// TIA Portal project "MersinKenet200_V18" (V18)

(* hardware
DEVICE "HMI_1"  KTP900 Basic PN
   slot 0: "HMI_1"  KTP900 Basic PN  6AV2 123-2JB03-0AX0  17.0.0.0
   slot 1: "HMI_RT_1"  KTP900 Basic PN  6AV2 123-2JB03-0AX0  17.0.0.0
   slot 5: "HMI_1.IE_CP_1"  PROFINET Interface  17.0.0.0
      slot 1: "PROFINET Interface_1"  PROFINET Interface
         slot 1: "Port_1"  Port
DEVICE "S7-1200 station_1"  S7-1200 Station
   slot 0: "Rack_0"  S7-1200 Rack  Rack  V1.0
   slot 1: "PLC_1"  CPU 1214C DC/DC/DC  6ES7 214-1AG40-0XB0  V4.5
   slot 2: "DI 16/DQ 16x24VDC_1"  6ES7 223-1BL32-0XB0  V2.0
DEVICE "GSD device_1"  GSD.Device.PN
   slot 0: "Rack"  Rack  V1.0
   slot 0: "SINAMICS-V90-PN"  SINAMICS V90 PN V1.0  6SL3 210-5Fxxx-xxFx  V1.00
      slot 0: "SINAMICS V90 PN V1.0"  SINAMICS V90 PN V1.0
      slot 1: "PN-IO"  PN-IO
         slot 1: "Port 1"  Port 1
         slot 2: "Port 2"  Port 2
      slot 1: "Drive_1"  Drive
         slot 0: "Module Access Point"  Module Access Point
         slot 1: "without PROFIsafe"  without PROFIsafe
   slot 2: "SIEMENS telegram 111, PZD-12/12"  SIEMENS telegram 111, PZD-12/12
DEVICE "GSD device_2"  GSD.Device.PN
   slot 0: "Rack"  Rack  V1.0
   slot 0: "CTEU-PN"  CTEU-PN  2201471
      slot 0: "CTEU-PN"  CTEU-PN
      slot 1: "PN-IO Interface"  PN-IO Interface
         slot 1: "Port 1"  Port 1
         slot 2: "Port 2"  Port 2
   slot 1: "VAEM-L1-S-8-PT_1"  VAEM-L1-S-8-PT  573384
      slot 0: "VAEM-L1-S-8-PT"  VAEM-L1-S-8-PT
*)

// ===== PLC "PLC_1"  CPU 1214C DC/DC/DC =====

VAR_GLOBAL   // PLC tag table "Default tag table"
   "System_Byte" AT %MB1 : Byte;
   "FirstScan" AT %M1.0 : Bool;
   "DiagStatusUpdate" AT %M1.1 : Bool;
   "AlwaysTRUE" AT %M1.2 : Bool;
   "AlwaysFALSE" AT %M1.3 : Bool;
   "ManVakum" AT %M4.7 : Bool;   // Vakum pedleri manuel kontrol
   "HaziraAl_P1_Ileri" AT %M2.0 : Bool;
   "HaziraAl_P1_Geri" AT %M2.1 : Bool;
   "HaziraAl_P2_Ileri" AT %M2.2 : Bool;
   "HaziraAl_P2_Geri" AT %M2.3 : Bool;
   "HaziraAl_P3_geri" AT %M3.0 : Bool;
   "HaziraAl_ServoGoPos" AT %M3.1 : Bool;
   "ClassA_Hazir" AT %M3.2 : Bool;
   "ClassF_Hazir" AT %M3.5 : Bool;
   "ClassE_Hazir" AT %M3.3 : Bool;
   "denemeStart" AT %M3.4 : Bool;   // denemeStart
   "m50.0" AT %M3.6 : Bool;   // empty
   "AcilStop_Ris" AT %M3.7 : Bool;
   "AcilStop_Fall" AT %M5.0 : Bool;
   "empty" AT %M22.0 : Bool;
   "AutoSeq_Yesil_Lamba_Durum1" AT %M5.1 : Bool;
   "Q0.2" AT %Q0.2 : Bool;   // kirmizi lamba
   "Q0.3" AT %Q0.3 : Bool;   // sari lamba
   "Q0.4" AT %Q0.4 : Bool;   // yesil lamba
   "Q0.5" AT %Q0.5 : Bool;   // vacum
   "Q0.6" AT %Q0.6 : Bool;   // Vinc aydinlatma
   "AutoSeq_Yesil_Lamba_Durum2" AT %M5.2 : Bool;
   "Bırakma_Pos" AT %MD6 : DInt;
   "Q0.0" AT %Q0.0 : Bool;
   "Q0.1" AT %Q0.1 : Bool;
   "Q4.0" AT %Q4.0 : Bool;   // P4B-geri(kenetleme)
   "Q4.1" AT %Q4.1 : Bool;   // P4B-ileri (kenetleme)
   "Q4.2" AT %Q4.2 : Bool;   // P4-geri (kenetleme)
   "Q4.3" AT %Q4.3 : Bool;   // P4-ileri (kenetleme)
   "Q4.4" AT %Q4.4 : Bool;   // P1-geri (enayar)
   "Q4.5" AT %Q4.5 : Bool;   // P1-ileri (enayar)
   "Q4.6" AT %Q4.6 : Bool;   // P2-geri (enayar)
   "Q4.7" AT %Q4.7 : Bool;   // P2-ileri (enayar)
   "Q5.0" AT %Q5.0 : Bool;   // P3-geri (kademe)
   "Q5.1" AT %Q5.1 : Bool;   // P3-ileri (kademe)
   "ManP2_EnAyar_Ileri" AT %M5.3 : Bool;
   "ManP2_EnAyar_Geri" AT %M5.4 : Bool;
   "Gerdirme_Pos" AT %MD10 : Real;
   "AutoSeq_P3_Ileri" AT %M5.5 : Bool;
   "ManServoGoPos2" AT %M5.6 : Bool;
   "btnStartForHmi" AT %M5.7 : Bool;
   "HaziraAl_P4_P4B_Geri" AT %M14.0 : Bool;
   "MemDrive_Standsill" AT %M14.1 : Bool;
   "HaziraAl_Started" AT %M14.2 : Bool;
   "I3.6" AT %I3.6 : Bool;   // uzak kontrol cift el 2/1
   "I3.7" AT %I3.7 : Bool;   // uzak kontrol cift el 2/2
   "RemoteCiftEl" AT %M14.3 : Bool;   // Uzak kumanda cift el butonları
   "ManKenetPisP4B_Ileri" AT %M14.4 : Bool;
   "ManKenetPisP4B_Geri" AT %M14.5 : Bool;
   "vakumJenRising" AT %M14.6 : Bool;
   "Falling_Vakum_Jen" AT %M14.7 : Bool;
   "Vakum_Edge" AT %M15.0 : Bool;
   "AlarmSustur" AT %M15.1 : Bool;
END_VAR

VAR_GLOBAL   // PLC tag table "PLC"
   "Clock_Byte" AT %MB0 : Byte;
   "Clock_10Hz" AT %M0.0 : Bool;
   "Clock_5Hz" AT %M0.1 : Bool;
   "Clock_2.5Hz" AT %M0.2 : Bool;
   "Clock_2Hz" AT %M0.3 : Bool;
   "Clock_1.25Hz" AT %M0.4 : Bool;
   "Clock_1Hz" AT %M0.5 : Bool;
   "Clock_0.625Hz" AT %M0.6 : Bool;
   "Clock_0.5Hz" AT %M0.7 : Bool;
END_VAR

VAR_GLOBAL   // PLC tag table "Manuel"
   "ManServoJog1" AT %M2.4 : Bool;   // Manuel servo jog 1
   "ManServoJog2" AT %M2.5 : Bool;   // Servo manuel jog 2
   "ManServoGoHome" AT %M2.6 : Bool;   // Servo manuel go home position
   "ManServoGoPos" AT %M2.7 : Bool;   // Servo manuel kenetleme pozisyonuna git
   "ManP1_EnAyar_Ileri" AT %M4.0 : Bool;   // Manuel en ayar pistonu ileri hareket
   "ManP1_EnAyar_Geri" AT %M4.1 : Bool;   // Manuel en ayar pistonu geri hareket
   "ManKenelemePisP4_Ileri" AT %M4.2 : Bool;   // Manuel kenetleme pistonu ileri hareket
   "ManKenelemePisP4_Geri" AT %M4.3 : Bool;   // Manuel kenetleme pistonu geri hareket
   "ManKademePisIleri" AT %M4.4 : Bool;   // Manuel kademe pistonu ileri hareket
   "ManKademePisGeri" AT %M4.5 : Bool;   // Manuel kademe pistonu geri hareket
   "ManVincLambasi" AT %M4.6 : Bool;   // Vinc lambası
END_VAR

VAR_GLOBAL   // PLC tag table "Peripheral"
   "I0.0" AT %I0.0 : Bool;   // Acil Stop
   "I0.1" AT %I0.1 : Bool;   // pizzato - Cift El
   "I0.2" AT %I0.2 : Bool;   // vakum tut-bırak 1
   "I0.3" AT %I0.3 : Bool;   // vakum tut-bırak 2
   "I0.4" AT %I0.4 : Bool;   // P1 ileride
   "I0.5" AT %I0.5 : Bool;   // p1 geride
   "I0.6" AT %I0.6 : Bool;   // p1a ileride
   "I0.7" AT %I0.7 : Bool;   // p1a geride
   "I1.0" AT %I1.0 : Bool;   // p2 ileride
   "I1.1" AT %I1.1 : Bool;   // p2 geride
   "I1.2" AT %I1.2 : Bool;   // p2a ileride
   "I1.3" AT %I1.3 : Bool;   // p2a geride
   "I1.4" AT %I1.4 : Bool;   // p3 ileride
   "I1.5" AT %I1.5 : Bool;   // p3 geride
   "I2.0" AT %I2.0 : Bool;   // p3a ileride
   "I2.1" AT %I2.1 : Bool;   // p3a geride
   "I2.2" AT %I2.2 : Bool;   // p4 ileride
   "I2.3" AT %I2.3 : Bool;   // p4 geride
   "I2.4" AT %I2.4 : Bool;   // p4a ileride
   "I2.5" AT %I2.5 : Bool;   // p4a geride
   "I2.6" AT %I2.6 : Bool;   // p4b ileride
   "I2.7" AT %I2.7 : Bool;   // p4b geride
   "I3.0" AT %I3.0 : Bool;   // p4c ileride
   "I3.1" AT %I3.1 : Bool;   // p4c geride
   "I3.2" AT %I3.2 : Bool;   // lamba butonu
END_VAR

TYPE "ReceiptModel"
   STRUCT
      "Name" : String[50];   // Model Adı - 50 karakter
      Class : Int;   // Model sınıfı ( A = 0, E= 1, F = 2 )
      Boy_C : Real := 500.0;   // Model boyu (C) - mm
      En_D : Real;   // Model eni (D) - mm
   END_STRUCT;
END_TYPE

// folder: Telegram111/Receive

TYPE "ZSW1"
   STRUCT
      TolError : Bool;   // ZSW1.8 1 = Following error within tolerance
      ControlReq : Bool;   // ZSW1.9 1 = Control requested
      TarPosReached : Bool;   // ZSW1.10 1 = Target position reached
      RefPointSet : Bool;   // ZSW1.11 1 = Reference point set
      TrvTskAck : Bool;   // ZSW1.12= Acknowledgement traversing block activated
      StndStill : Bool;   // ZSW1.13 1 = This bit is used for standstill detection
      AxisAcc : Bool;   // ZSW1.14 1 = Axis accelerated
      AxisDec : Bool;   // ZSW1.15 1 = Axis decelerated
      RTS : Bool;   // ZSW1.0 1 =Ready to power up
      RDY : Bool;   // ZSW1.1 1 = Ready for operation (DC link loaded, pulses blocked)
      IOp : Bool;   // ZSW1.2 1 = Drive is switched on
      Fault : Bool;   // ZSW1.3 1 = Fault present
      OFF2Inactive : Bool;   // ZSW1.4 1 = No coast down active (OFF2 inactive)
      OFF3Inactive : Bool;   // ZSW1.5 1 = No fast stop active (OFF3 inactive)
      PowInhbt : Bool;   // ZSW1.6 1 = Activation disable active
      Alarm : Bool;   // ZSW1.7 1 = Alarm present
   END_STRUCT;
END_TYPE

TYPE "POS_ZSW1"
   STRUCT
      StopCamAct : Bool := FALSE;   // (POS_ZSW1.8) - 1 = STOP cam minus active
      StopCamPlusAct : Bool := FALSE;   // (POS_ZSW1.9) - 1 = STOP cam plus active
      jogActive : Bool := FALSE;   // (POS_ZSW1.10) - 1 = Jogging active
      ReferencePointAct : Bool := FALSE;   // (POS_ZSW1.11) - 1 = Reference point approach active
      FlyRefAct : Bool := FALSE;   // (POS_ZSW1.12) - On-the-fly homing active
      TrvBlockAct : Bool := FALSE;   // (POS_ZSW1.13) - 1 = Traversing Block active
      MdiStupAct : Bool := FALSE;   // (POS_ZSW1.14) - 1 = Set-up active
      MdiPosAct : Bool := FALSE;   // (POS_ZSW1.15) - 1 = MDI active
      Reserve : Byte;
   END_STRUCT;
END_TYPE

TYPE "POS_ZSW2"
   STRUCT
      PosActLowerCam : Bool := FALSE;   // (POS_ZSW2.8) - 1 = Position actual value ≤ cam switching position 1
      PosActGreaterCam : Bool := FALSE;   // (POS_ZSW2.9) - 1 = Position actual value ≤ cam switching position 2
      DirOut1 : Bool := FALSE;   // (POS_ZSW2.10) - 1 = Direct output 1 via traversing block
      DirOut2 : Bool := FALSE;   // (POS_ZSW2.11) - 1 = Direct output 2 via traversing block
      FixStopReached : Bool := FALSE;   // (POS_ZSW2.12) - 1 = Fixed stop reached
      FixStopTorque : Bool := FALSE;   // (POS_ZSW2.13) - 1 = Fixed stop clamping torque reached
      TravelToFixStopAct : Bool := FALSE;   // (POS_ZSW2.14) - 1 = Travel to fixed stop active
      TraversingAct : Bool := FALSE;   // (POS_ZSW2.15) - 1 = Traversing command active
      TrackingModeAct : Bool := FALSE;   // (POS_ZSW2.0) 1 = Tracking mode active
      VelocityLimAct : Bool := FALSE;   // (POS_ZSW2.1) - 1 = Velocity limiting active
      SetPStat : Bool := FALSE;   // (POS_ZSW2.2) - 1 = Setpoint set
      reserv : Bool := FALSE;   // (POS_ZSW2.3) - reserved
      MovesForward : Bool := FALSE;   // (POS_ZSW2.4) - 1 = Axis moves forward
      MovesBackward : Bool := FALSE;   // (POS_ZSW2.5) - 1 = Axis moves backwards
      SftLimSwMinReached : Bool := FALSE;   // (POS_ZSW2.6) - 1 = Software limit switch minus reached
      SftLimSwPlusReached : Bool := FALSE;   // (POS_ZSW2.7) - 1 = Software limit switch plus reached
   END_STRUCT;
END_TYPE

TYPE "ZSW2"
   STRUCT
      Reserve : Byte;
      Reserve_1 : Byte;
   END_STRUCT;
END_TYPE

TYPE "MELDW"
   STRUCT
      SpeedSetPoint : Bool;   // 1 = Speed setpoint - actual value deviation within tolerance t_on
      Reserv : Bool;
      Reserv_1 : Bool;
      ControllerEn : Bool;   // 1 = Controller enable
      DriveReady : Bool;   // MELDW.12 - 1 = Drive ready
      PulseEn : Bool;   // MELDW.13 1 = Pulses enabled
      Reserv_2 : Bool;
      Reserv_3 : Bool;
      RampFuncAct : Bool;   // MELDW.0 1 = Ramp-up/ramp-down complete 0 = Ramp-function generator active
      Reserv_4 : Bool;
      Reserv_5 : Bool;
      Reserv_6 : Bool;
      Reserv_7 : Bool;
      Reserv_8 : Bool;
      NoMotOverTemp : Bool;   // MELDW.6 1 = No motor overtemperature alarm
      NoAlrmOverload : Bool;   // MELDW.7 1 = No alarm, thermal overload, power unit
   END_STRUCT;
END_TYPE

// folder: Telegram111/Send

TYPE "STW1"
   STRUCT
      Jog1 : Bool;   // (STW1.8) - Jog 1 signal source
      Jog2 : Bool;   // (STW1.9) - Jog 2 signal source
      ControlByPlc : Bool;   // (STW1.10) - 1 = Control via PLC
      RefStart : Bool;   // (STW1.11) - 1 = Start referencing
      reserved : Bool;
      ExtBlockChange : Bool;
      reserved_1 : Bool;
      reserved_2 : Bool;
      Off1 : Bool;   // (STW1.0) - ON - 0 = OFF1 active; 1 = ON
      Off2 : Bool;   // (STW1.1) - 1 = Operating condition no coast down active
      Off3 : Bool;   // (STW1.2) - 1 = Operating condition no quick stop active
      InverterEn : Bool;   // (STW1.3) - 1 = Inverter enable
      RjcTraverTask : Bool;   // (STW1.4) - 1 = Do not reject traversing task
      IndStop : Bool;   // (STW1.5) - 1 = No intermediate stop
      TrvStart : Bool;   // (STW1.6) - Activate traversing task
      AckFaults : Bool;   // (STW1.7) - Acknowledge faults
   END_STRUCT;
END_TYPE

TYPE "POS_STW1"
   STRUCT
      MdiType : Bool;   // (POS_STW1.8) - 1 = Absolute positioning is selected 0 = Relative positioning is selected
      MdiPos : Bool;   // (POS_STW1.9) Direction selection for setting up or absolute positioning
      MdiNeg : Bool;   // (POS_STW1.10) Direction selection for setting up or absolute positioning
      reserv : Bool;
      MdiTrType : Bool;   // (POS_STW1.12) 0 = Applying values by rising edge on MdiEdge 1 = Signal: constant setpoint transfer
      reserv_1 : Bool;
      MdiSetup : Bool;   // (POS_STW1.14) => 0 = Position 1 = Setup
      MdiStart : Bool;   // (POS_STW1.15) => Operating mode MDI / direct setpoint specification
      Reserved : Byte;   // Traversing bock selection vb.
   END_STRUCT;
END_TYPE

TYPE "POS_STW2"
   STRUCT
      RefType : Bool;   // (POS_STW2.8) Homing type selection 0 = Reference point approach 1 = On-the-fly homing
      RefStartDir : Bool;   // (POS_STW2.9) - 1 = Start the search for reference in the negative direction0 = Start the search for reference in the positive direction
      RefInpS : Bool;
      RefEdge : Bool;   // (POS_STW2.11) passive homing: Setting the edge evaluation 0 = rising edge 1 = falling edge
      Reserv_3 : Bool;
      Reserv_4 : Bool;
      SftLimAct : Bool;   // (POS_STW2.14) - 1= Software limit switch activation
      StopCamAct : Bool;   // (POS_STW2.15) -1 = STOP cam active
      TrakingModeActive : Bool;   // (POS_STW2.0) -1 = Tracking mode active
      SetRefPoint : Bool;   // (POS_STW2.1) -1 = Set reference point
      ActRefCam : Bool;   // (POS_STW2.2) -1 = Reference cam active
      Reserv_5 : Bool;
      Reserv_6 : Bool;
      JogIncActv : Bool;   // (POS_STW2.5) => 0 = Continuous procedure 1 = Procedure by parameterized path
      Reserv_7 : Bool;
      Reserv_8 : Bool;
   END_STRUCT;
END_TYPE

TYPE "STW2"
   STRUCT
      Reserv : Byte;
      Reserv_1 : Byte;
   END_STRUCT;
END_TYPE

// folder: Alarm

DATA_BLOCK "Alarm_DB"   // DB9
{ S7_Optimized_Access := 'TRUE' }
VERSION : 0.1
// stored: InstanceOfName Alarm
"Alarm"
BEGIN
END_DATA_BLOCK

// folder: General

DATA_BLOCK "Out_DB"   // DB2
{ S7_Optimized_Access := 'TRUE' }
VERSION : 0.1
// stored: InstanceOfName InOut
"InOut"
BEGIN
END_DATA_BLOCK

DATA_BLOCK "HMI_Data"   // DB5
{ S7_Optimized_Access := 'TRUE' }
VERSION : 0.1
   VAR
      btnStart : Bool;
      btnStop : Bool;
      btnManuel : Bool;
      btnAuto : Bool;
      btnHaziraAl : Bool;
      EnAyarPistonu : Struct   // P1 - P2
         P1 : Struct
            btnIleri : Bool;
            btnGeri : Bool;
         END_STRUCT;
         P2 : Struct
            btnIleri : Bool;
            btnGeri : Bool;
         END_STRUCT;
      END_STRUCT;
      KenetlemePistonu : Struct   // P4-P4B
         P4 : Struct   // SAG KOLON KENETLEME
            btnIleri : Bool;
            btnGeri : Bool;
         END_STRUCT;
         P4B : Struct   // SOL KOLON KENETLEME
            btnIleri : Bool;
            btnGeri : Bool;
         END_STRUCT;
      END_STRUCT;
      "Kademe Pistonu" : Struct   // P3
         btnIleri : Bool;
         btnGeri : Bool;
      END_STRUCT;
      btnVincLambasi : Bool;
      ServoButton : Struct
         btnJogIleri : Bool;
         btnJogGeri : Bool;
         btnRefNokBelirle : Bool;
         btnHome : Bool;
         btnGoPos : Bool;
         btnHataReset : Bool;
         btnStop : Bool;   // Servo manuel işlemini durdur
         btnKenetle : Bool;   // kenetleme pozisyonuna git
      END_STRUCT;
   END_VAR
   VAR RETAIN
      ServoData : Struct
         txtActPozisyon : Real;
         txtJogOverride : Int := 100;
         txtVelocity : Real := 50.0;
         txtGerdirmeMes : Real := 10.0;   // parca gerdirme mesafesi
      END_STRUCT;
   END_VAR
   VAR
      MainInfo : String[50];
      ServoInfo : String[40];
   END_VAR
   VAR RETAIN
      KenetlemeSuresi : Time := T#1s;
   END_VAR
   VAR
      Buttons : Struct
         btnVakumJeneratoru : Bool;
         btnAlarmSustur : Bool;
      END_STRUCT;
      Status : Struct
         EnAyarPis : Struct   // P1-P1A-P2-P2A pistonları
            P1 : Struct
               Ileride : Bool;   // P1-P1A ileride
               Geride : Bool;   // P1-P1A geride
            END_STRUCT;
            P2 : Struct
               Ileride : Bool;   // P2-P2A ileride
               Geride : Bool;   // P2-P2A geride
            END_STRUCT;
         END_STRUCT;
         KademePis_P3 : Struct   // P3 pistonu
            Ileride : Bool;   // P3 pistonu ileride
            Geride : Bool;   // P3 pistonu geride
         END_STRUCT;
         KenetlemePis_P4 : Struct   // P4-P4B pistonları
            Ileride : Bool;   // P4-P4B pistonları ileride
            Geride : Bool;   // P4-P4B pistonları geride
         END_STRUCT;
      END_STRUCT;
      Alarms : Word;
      AcilSayfasi : Bool;
   END_VAR
BEGIN
END_DATA_BLOCK

DATA_BLOCK "Peripheral_Data"   // DB6
{ S7_Optimized_Access := 'TRUE' }
VERSION : 0.1
   VAR
      IN : Struct
         Acil_Stop : Bool;
         CiftEl : Struct
            IN1 : Bool;   // pizzato cift el
            IN2 : Bool;   // remote cift el 1
            IN3 : Bool;   // remote cift el 2
         END_STRUCT;
         EnAyar : Struct   // P1,P1A,P2,P2A
            P1 : Struct
               Ileride : Bool;
               Geride : Bool;
            END_STRUCT;
            P1A : Struct
               Ileride : Bool;
               Geride : Bool;
            END_STRUCT;
            P2 : Struct
               Ileride : Bool;
               Geride : Bool;
            END_STRUCT;
            P2A : Struct
               Ileride : Bool;
               Geride : Bool;
            END_STRUCT;
         END_STRUCT;
         KademeAyar : Struct   // P3,P3A
            P3 : Struct
               Ileride : Bool;
               Geride : Bool;
            END_STRUCT;
         END_STRUCT;
         Kenetleme : Struct   // P4,P4A,P4B,P4C
            P4 : Struct
               Ilderide : Bool;
               Geride : Bool;
            END_STRUCT;
            P4B : Struct
               Ilderide : Bool;
               Geride : Bool;
            END_STRUCT;
         END_STRUCT;
         VincUstuLamba : Bool;
         VakumJen : Bool;
         ServoHomeSen : Bool;   // Servo home sensoru
      END_STRUCT;
      OUT : Struct
         EnAyar : Struct   // P1,P1A,P2,P2A
            P1 : Struct
               Ileri : Bool;
               Geri : Bool;
            END_STRUCT;
            P2 : Struct
               Ileri : Bool;
               Geri : Bool;
            END_STRUCT;
         END_STRUCT;
         KademeAyar : Struct   // P3,P3A
            P3 : Struct
               Ileri : Bool;
               Geri : Bool;
            END_STRUCT;
         END_STRUCT;
         Kenetleme : Struct   // P4,P4A,P4B,P4C
            P4_P4A : Struct
               Ilderi : Bool;
               Geri : Bool;
            END_STRUCT;
            P4B_P4C : Struct
               Ilderi : Bool;
               Geri : Bool;
            END_STRUCT;
         END_STRUCT;
         LAMBA : Struct
            Yesil : Bool;
            Kirmizi : Bool;
            Sari : Bool;
            Buzzer : Bool;
         END_STRUCT;
         VincLambasi : Bool;
         Vacum : Bool;   // Vakum jeneratoru
      END_STRUCT;
   END_VAR
BEGIN
END_DATA_BLOCK

DATA_BLOCK "System_Data"   // DB7
{ S7_Optimized_Access := 'TRUE' }
VERSION : 0.1
   VAR
      AutoSeq_State : Int;
      AutoSeq_Busy : Bool;
      AutoSeq_Done : Bool;
      AutoSeq_Message : String[50];
      Ready : Bool;
      CmdDrive : Struct
         GoPos : Bool;
         GoHome : Bool;
         SetReference : Bool;
         Jog1 : Bool;
         Jog2 : Bool;
         Position : Real;
         Velocity : Real;
         Override : Int;
         AckError : Bool;
         Message : String[40];
         Pos_Done : Bool;
         Busy : Bool;
         Error : Bool;
         AxisError : Bool;
         ErrorId : Byte;
         ReferencedAxis : Bool;
         ActPosition : Real;
         HomePosition : Real;   // Servo durması gereken home pozisyonu
         Alarm : Word;
         IsHomePosTol : Bool;   // Axis home konumu tolerans icinde
         IsPosTol : Bool;   // Axis pozisyon konumu tolerans icinde
      END_STRUCT;
      SystemMode : Struct
         Auto : Bool;
         Man : Bool;
      END_STRUCT;
      AutoSeq : Struct
         GoPos : Bool;   // Parça kenetleme
         GoPos2 : Bool;   // Parça birakma
         GoHome : Bool;
         P3_Ileri : Bool;
         P3_Geri : Bool;   // kademe pistonu
         "P4-P4A_Ileri" : Bool;   // kenetleme pistonu
         "P4-P4A_geri" : Bool;
         "P4B-P4C_Ileri" : Bool;
         StartedInfo : Bool;   // otomatik mod basladi
      END_STRUCT;
   END_VAR
BEGIN
END_DATA_BLOCK

DATA_BLOCK "SINA_POS_DB"   // DB11
{ S7_Optimized_Access := 'TRUE' }
AUTHOR : DRVDPS7
FAMILY : DRIVES
NAME : SINA_POS
VERSION : 5.7
// stored: InstanceOfName SINA_POS
"SINA_POS"
BEGIN
END_DATA_BLOCK

// folder: Manuel

DATA_BLOCK "Manuel_DB"   // DB4
{ S7_Optimized_Access := 'TRUE' }
VERSION : 0.1
// stored: InstanceOfName Manuel
"Manuel"
BEGIN
END_DATA_BLOCK

// folder: Otomatik

DATA_BLOCK "Otomatik_Seq_LAD_DB"   // DB8
{ S7_Optimized_Access := 'TRUE' }
VERSION : 0.1
// stored: InstanceOfName Otomatik_Seq_LAD
"Otomatik_Seq_LAD"
BEGIN
END_DATA_BLOCK

// folder: Receipt

DATA_BLOCK "Receipt"   // DB1
{ S7_Optimized_Access := 'TRUE' }
VERSION : 0.1
   VAR RETAIN
      ModelId : Int;   // Combobox index numarasi
      OldModelId : Int;
      ModelList : Array[0..25] of "ReceiptModel";   // Model listesi
      CurrentModel : "ReceiptModel";   // Secili model
   END_VAR
   VAR
      btnSave : Bool;   // Recete kaydet butonu - HMI
      bShowMessage : Bool;   // Kaydedildi mesaji icin
      tSavedTimer : IEC_TIMER;
   END_VAR
BEGIN
END_DATA_BLOCK

// folder: (top level)

ORGANIZATION_BLOCK "Task_1"   // OB1, LAD, ProgramCycle
TITLE = "Main Program Sweep (Cycle)"
{ S7_Optimized_Access := 'TRUE' }
VERSION : 0.1
   VAR_INPUT
      Initial_Call : Bool;   // Initial call of this OB
      Remanence : Bool;   // =True, if remanent data are available
   END_VAR
   VAR_TEMP
      bSeqStart : Bool;   // Otomatik sekans baslat
   END_VAR
BEGIN

REGION Network 1: Sistem acildiginda ilk cycle ile manuel setle (bir seferlik calisir)
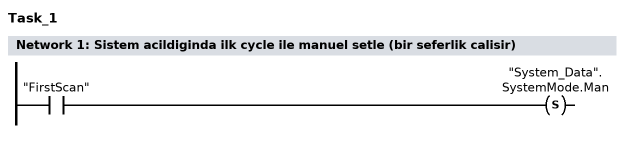
   RUNG wire#powerrail
      Contact( "FirstScan" )
      S_Coil( "System_Data".SystemMode.Man )
   END_RUNG
   // the same network as SCL:
   IF "FirstScan" THEN "System_Data".SystemMode.Man := TRUE; END_IF;
END_REGION

REGION Network 2 (SCL): Otomatik sekans baslat
   "Peripheral"();
   "Out_DB"();
   "Station"();

   #bSeqStart := "Peripheral_Data".IN.CiftEl.IN1 AND "RemoteCiftEl";
   "Otomatik_Seq_LAD_DB"(Start := #bSeqStart,
                         //Start := "btnStartForHmi",
                         Stop := "HMI_Data".btnStop,
                         EmergencyStop := "Peripheral_Data".IN.Acil_Stop,
                         Busy => "System_Data".AutoSeq_Busy,
                         Done => "System_Data".AutoSeq_Done,
                         Message => "System_Data".AutoSeq_Message);
END_REGION
END_ORGANIZATION_BLOCK

ORGANIZATION_BLOCK "Hardware interrupt"   // OB40, LAD, HWProcessInterrupt
{ S7_Optimized_Access := 'TRUE' }
VERSION : 0.1
   VAR_INPUT
      LADDR : Hw_Io;   // Hardware identifier
      USI : Word;   // User structure identifier
      IChannel : USInt;   // Interrupt channel number
      EventType : Byte;   // EventType
   END_VAR
BEGIN
END_ORGANIZATION_BLOCK

ORGANIZATION_BLOCK "Diagnostic error interrupt"   // OB82, LAD, DiagnosticErrorInterrupt
{ S7_Optimized_Access := 'TRUE' }
VERSION : 0.1
   VAR_INPUT
      IO_State : Word;   // IO state of the HW object
      LADDR : Hw_Any;   // Hardware identifier
      Channel : UInt;   // Channel number
      MultiError : Bool;   // =true if more than one error is present
   END_VAR
BEGIN
END_ORGANIZATION_BLOCK

ORGANIZATION_BLOCK "Pull or plug of modules"   // OB83, LAD, PullPlug
{ S7_Optimized_Access := 'TRUE' }
VERSION : 0.1
   VAR_INPUT
      LADDR : Hw_Io;   // Hardware identifier
      Event_Class : Byte;   // 16#38/39: module inserted, removed
      Fault_ID : Byte;   // Fault identifier
   END_VAR
BEGIN
END_ORGANIZATION_BLOCK

ORGANIZATION_BLOCK "Rack or station failure"   // OB86, LAD, RackStationFailure
{ S7_Optimized_Access := 'TRUE' }
VERSION : 0.1
   VAR_INPUT
      LADDR : Hw_Device;   // Hardware identifier
      Event_Class : Byte;   // Event class
      Fault_ID : Byte;   // Fault identifier
   END_VAR
BEGIN
END_ORGANIZATION_BLOCK

ORGANIZATION_BLOCK "Startup"   // OB100, LAD, Startup
TITLE = "Complete Restart"
{ S7_Optimized_Access := 'TRUE' }
VERSION : 0.1
   VAR_INPUT
      LostRetentive : Bool;   // True if retentive data are lost
      LostRTC : Bool;   // True if date and time are lost
   END_VAR
BEGIN

REGION Network 1
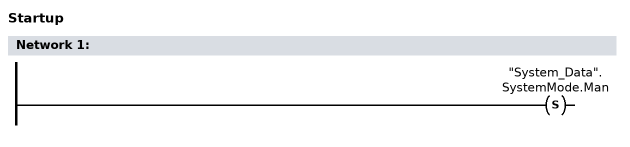
   RUNG wire#powerrail
      S_Coil( "System_Data".SystemMode.Man )
   END_RUNG
   // the same network as SCL:
   "System_Data".SystemMode.Man := TRUE;
END_REGION
END_ORGANIZATION_BLOCK

ORGANIZATION_BLOCK "Task_2"   // OB123, LAD, ProgramCycle
TITLE = "Main Program Sweep (Cycle)"
{ S7_Optimized_Access := 'TRUE' }
VERSION : 0.1
   VAR_INPUT
      Initial_Call : Bool;   // Initial call of this OB
      Remanence : Bool;   // =True, if remanent data are available
   END_VAR
BEGIN

REGION Network 2 (SCL)
   "ReceiptManager"();
   "Manuel_DB"();
   "HMI"();
   "HaziraAl"(Execute:="HMI_Data".btnHaziraAl,
              EmergencyStop:="Peripheral_Data".IN.Acil_Stop,
              IsServoPosDone:="System_Data".CmdDrive.Pos_Done,
              Manuel:="System_Data".SystemMode.Man,
              AxisReferenced:="System_Data".CmdDrive.ReferencedAxis,
              P1_Ileri=>"HaziraAl_P1_Ileri",
              P1_Geri=>"HaziraAl_P1_Geri",
              P2_Ileri=>"HaziraAl_P2_Ileri",
              P2_geri=>"HaziraAl_P2_Geri",
              P3_geri=>"HaziraAl_P3_geri",
              P4_P4B_Geri=>"HaziraAl_P4_P4B_Geri",
              ServoGoPos=>"HaziraAl_ServoGoPos",
              ClassA_Hazir=>"ClassA_Hazir",
              ClassE_Hazir=>"ClassE_Hazir",
              ClassF_Hazir=>"ClassF_Hazir");

   "Alarm_DB"();
   "UyariLambasi"();
END_REGION
END_ORGANIZATION_BLOCK

// folder: Alarm

FUNCTION_BLOCK "Alarm"   // FB7, LAD
{ S7_Optimized_Access := 'TRUE' }
VERSION : 0.1
   VAR
      timeInterval : Time;
      p1_ileri_Timer : TON_TIME;
      p1_geri_Timer : TON_TIME;
      p2_Ileri_Timer : TON_TIME;
      p2_geri_Timer : TON_TIME;
      p3_ileri_Timer : TON_TIME;
      p3_geri_Timer : TON_TIME;
      p4_ileri_Timer : TON_TIME;
      p4_geri_Timer : TON_TIME;
      p4b_ileri_Timer : TON_TIME;
      p4b_geri_Timer : TON_TIME;
      wAlarmsServoOrCylinder : Word;
      wAlarmsPeripheral : Word;
   END_VAR
BEGIN

REGION Network 1: timer interval
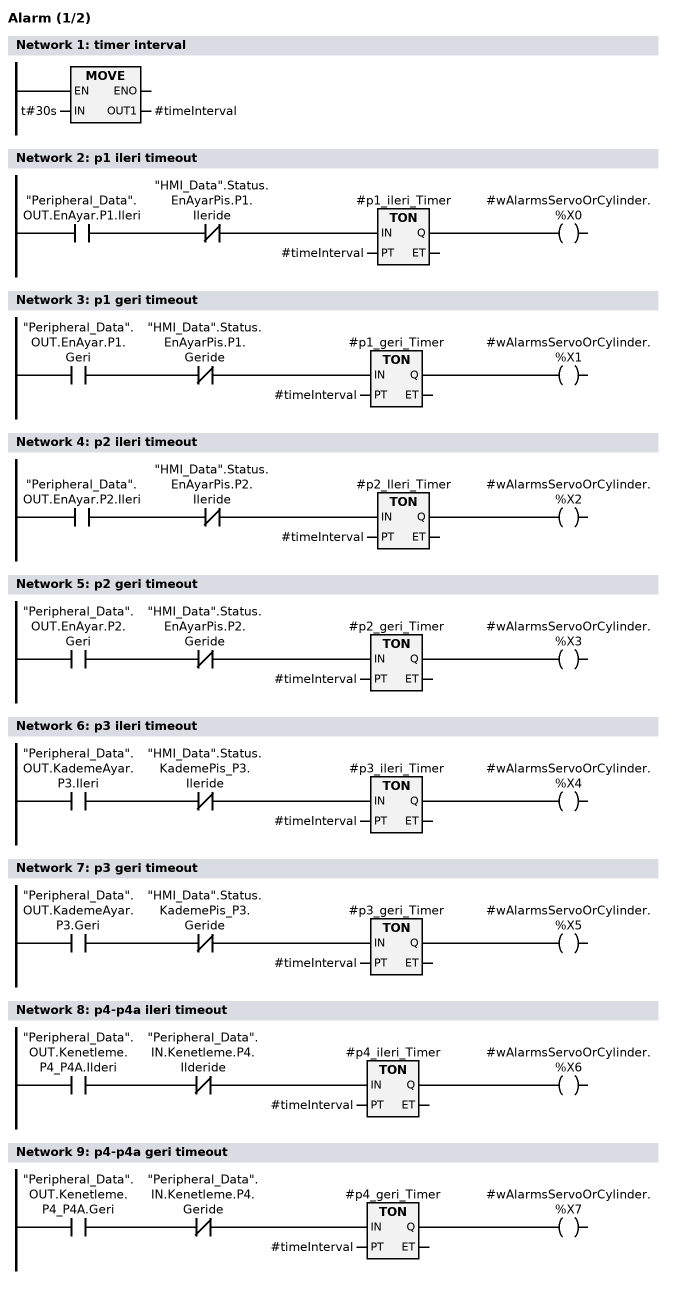
   RUNG wire#powerrail
      Move(in := t#30s, out1 => #timeInterval)
   END_RUNG
   // the same network as SCL:
   #timeInterval := t#30s;
END_REGION

REGION Network 2: p1 ileri timeout
   #p1_ileri_Timer(IN := "Peripheral_Data".OUT.EnAyar.P1.Ileri AND NOT "HMI_Data".Status.EnAyarPis.P1.Ileride,   // TON
                   PT := #timeInterval);
   #wAlarmsServoOrCylinder.%X0 := #p1_ileri_Timer.Q;
END_REGION

REGION Network 3: p1 geri timeout
   #p1_geri_Timer(IN := "Peripheral_Data".OUT.EnAyar.P1.Geri AND NOT "HMI_Data".Status.EnAyarPis.P1.Geride,   // TON
                  PT := #timeInterval);
   #wAlarmsServoOrCylinder.%X1 := #p1_geri_Timer.Q;
END_REGION

REGION Network 4: p2 ileri timeout
   #p2_Ileri_Timer(IN := "Peripheral_Data".OUT.EnAyar.P2.Ileri AND NOT "HMI_Data".Status.EnAyarPis.P2.Ileride,   // TON
                   PT := #timeInterval);
   #wAlarmsServoOrCylinder.%X2 := #p2_Ileri_Timer.Q;
END_REGION

REGION Network 5: p2 geri timeout
   #p2_geri_Timer(IN := "Peripheral_Data".OUT.EnAyar.P2.Geri AND NOT "HMI_Data".Status.EnAyarPis.P2.Geride,   // TON
                  PT := #timeInterval);
   #wAlarmsServoOrCylinder.%X3 := #p2_geri_Timer.Q;
END_REGION

REGION Network 6: p3 ileri timeout
   #p3_ileri_Timer(IN := "Peripheral_Data".OUT.KademeAyar.P3.Ileri AND NOT "HMI_Data".Status.KademePis_P3.Ileride,   // TON
                   PT := #timeInterval);
   #wAlarmsServoOrCylinder.%X4 := #p3_ileri_Timer.Q;
END_REGION

REGION Network 7: p3 geri timeout
   #p3_geri_Timer(IN := "Peripheral_Data".OUT.KademeAyar.P3.Geri AND NOT "HMI_Data".Status.KademePis_P3.Geride,   // TON
                  PT := #timeInterval);
   #wAlarmsServoOrCylinder.%X5 := #p3_geri_Timer.Q;
END_REGION

REGION Network 8: p4-p4a ileri timeout
   #p4_ileri_Timer(IN := "Peripheral_Data".OUT.Kenetleme.P4_P4A.Ilderi AND NOT "Peripheral_Data".IN.Kenetleme.P4.Ilderide,   // TON
                   PT := #timeInterval);
   #wAlarmsServoOrCylinder.%X6 := #p4_ileri_Timer.Q;
END_REGION

REGION Network 9: p4-p4a geri timeout
   #p4_geri_Timer(IN := "Peripheral_Data".OUT.Kenetleme.P4_P4A.Geri AND NOT "Peripheral_Data".IN.Kenetleme.P4.Geride,   // TON
                  PT := #timeInterval);
   #wAlarmsServoOrCylinder.%X7 := #p4_geri_Timer.Q;
END_REGION

REGION Network 10: p4b-p4c ileri timeout
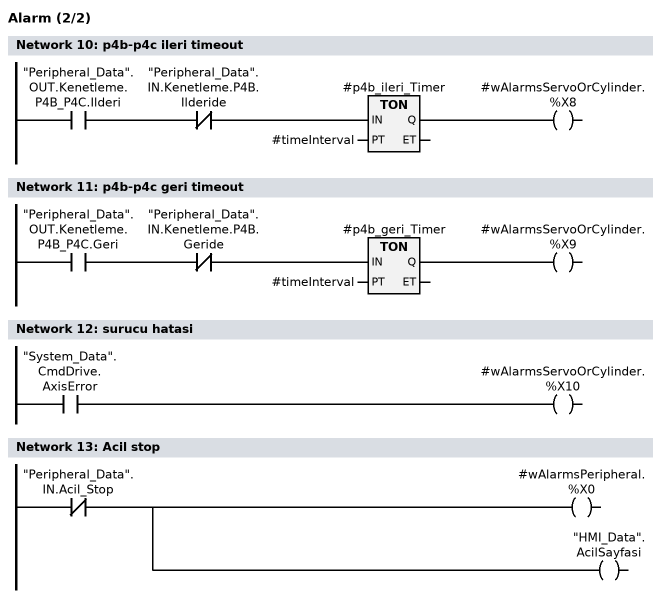
   #p4b_ileri_Timer(IN := "Peripheral_Data".OUT.Kenetleme.P4B_P4C.Ilderi AND NOT "Peripheral_Data".IN.Kenetleme.P4B.Ilderide,   // TON
                    PT := #timeInterval);
   #wAlarmsServoOrCylinder.%X8 := #p4b_ileri_Timer.Q;
END_REGION

REGION Network 11: p4b-p4c geri timeout
   #p4b_geri_Timer(IN := "Peripheral_Data".OUT.Kenetleme.P4B_P4C.Geri AND NOT "Peripheral_Data".IN.Kenetleme.P4B.Geride,   // TON
                   PT := #timeInterval);
   #wAlarmsServoOrCylinder.%X9 := #p4b_geri_Timer.Q;
END_REGION

REGION Network 12: surucu hatasi
   RUNG wire#powerrail
      Contact( "System_Data".CmdDrive.AxisError )
      Coil( #wAlarmsServoOrCylinder.%X10 )
   END_RUNG
   // the same network as SCL:
   #wAlarmsServoOrCylinder.%X10 := "System_Data".CmdDrive.AxisError;
END_REGION

REGION Network 13: Acil stop
   RUNG wire#powerrail
      I_Contact( "Peripheral_Data".IN.Acil_Stop )
      wire#w1
      Coil( #wAlarmsPeripheral.%X0 )
   END_RUNG
   RUNG wire#w1
      Coil( "HMI_Data".AcilSayfasi )
   END_RUNG
   // the same network as SCL:
   #wAlarmsPeripheral.%X0 := NOT "Peripheral_Data".IN.Acil_Stop;
   "HMI_Data".AcilSayfasi := NOT "Peripheral_Data".IN.Acil_Stop;
END_REGION
END_FUNCTION_BLOCK

// folder: BaseClass

FUNCTION_BLOCK "CiftEl"   // FB11, LAD
{ S7_Optimized_Access := 'TRUE' }
VERSION : 0.1
   VAR_INPUT
      In_1 : Bool;   // Cift el
      In_2 : Bool;   // Cift el
   END_VAR
   VAR_OUTPUT
      Out : Bool;   // out
   END_VAR
   VAR
      IEC_Timer_0_Instance : TP_TIME;
      IEC_Timer_0_Instance_1 : TP_TIME;
      IEC_Timer_0_Instance_2 : TOF_TIME;
      stOut : Bool;
   END_VAR
   VAR_TEMP
      bCiftEl_1 : Bool;
      bCiftEl_2 : Bool;
   END_VAR
BEGIN

REGION Network 1
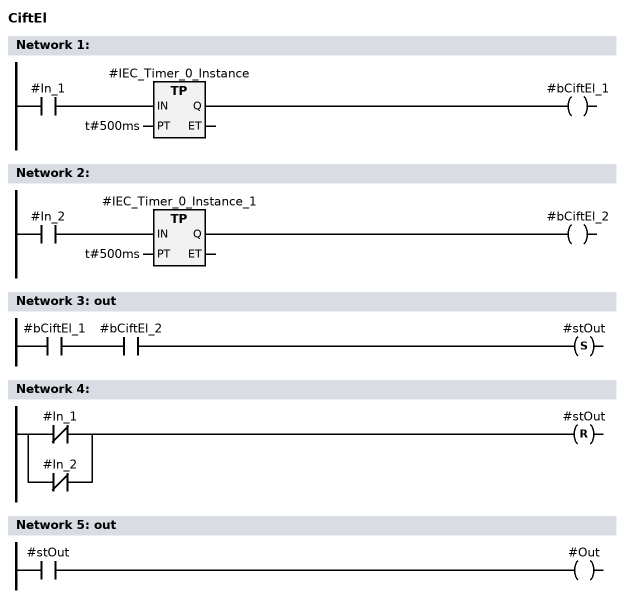
   #IEC_Timer_0_Instance(IN := #In_1, PT := t#500ms);   // TP
   #bCiftEl_1 := #IEC_Timer_0_Instance.Q;
END_REGION

REGION Network 2
   #IEC_Timer_0_Instance_1(IN := #In_2, PT := t#500ms);   // TP
   #bCiftEl_2 := #IEC_Timer_0_Instance_1.Q;
END_REGION

REGION Network 3: out
   RUNG wire#powerrail
      Contact( #bCiftEl_1 )
      Contact( #bCiftEl_2 )
      S_Coil( #stOut )
   END_RUNG
   // the same network as SCL:
   IF #bCiftEl_1 AND #bCiftEl_2 THEN #stOut := TRUE; END_IF;
END_REGION

REGION Network 4
   RUNG wire#powerrail
      I_Contact( #In_1 )
      wire#w1
      R_Coil( #stOut )
   END_RUNG
   RUNG wire#powerrail
      I_Contact( #In_2 )
   END_RUNG wire#w1
   // the same network as SCL:
   IF NOT #In_1 OR NOT #In_2 THEN #stOut := FALSE; END_IF;
END_REGION

REGION Network 5: out
   RUNG wire#powerrail
      Contact( #stOut )
      Coil( #Out )
   END_RUNG
   // the same network as SCL:
   #Out := #stOut;
END_REGION
END_FUNCTION_BLOCK

// folder: BaseClass/Drive

FUNCTION_BLOCK "BaseDrive_LAD"   // FB10, LAD
{ S7_Optimized_Access := 'TRUE' }
VERSION : 0.1
   VAR_INPUT
      Enable : Bool;   // BaseDrive enable
      Emergency : Bool;   // acil stop
      GoPos : Bool;   // kenetleme pozisyonuna git
      SetReference : Bool;   // referans ayarla
      Jog1 : Bool;   // servo jog 1 - negatif yon
      Jog2 : Bool;   // servo jog 1 - positive yon
      Position : Real;   // model kenetleme konumu
      Velocity : Real := 50.0;   // % (0 - 100) arası
      Override : Int := 100;   // % (0 - 100) arası
      AckError : Bool;   // servo hata reset
      HWDSTW : Hw_Io;
      HWDZSW : Hw_Io;
   END_VAR
   VAR_OUTPUT
      Pos_Done : Bool;
      Busy : Bool;
      Error : Bool;
      AxisError : Bool;   // Axis hatasi
      ErrorId : Byte;
      ReferencedAxis : Bool;   // reference point set
      Message : String[40];
      ActPosition : Real;
      Alarm : Word;   // Drive hataları
      IsPosTol : Bool;   // Axis pozisyon konumu tolerans icinde
      Standstill : Bool;   // servo durdu
   END_VAR
   VAR
      SINA_POS_Instance_1 : "SINA_POS";
      stState : Int;
      stMdiMode : Int;
      stEnableAxis : Bool;
      stTargetPos : DInt;
      stVelocity : DInt;
      stExecute : Bool;
      stAxisPosDone : Bool;
      stAxisError : Bool;
      IsDoneDelay : TON_TIME;
      DelayMessage : TON_TIME;
      IsDoneDelay_IN : Bool;
      IsDoneDelay_Q : Bool;
      DelayMessage_IN : Bool;
      DelayMessage_Q : Bool;
      stOverride : Int;
      stActualPosition : DInt;
      stHomingMode : Int;
      stHomingError : Bool;
      stHomingErrorId : Word;
      bHomingRefOk : Bool;
      stActualVelocity : DInt;
      DelayOnOff1_1 : TON_TIME;
      DelayOnOff1_2 : TON_TIME;
      DelayOnOff1_1_IN : Bool;
      DelayOnOff1_1_Q : Bool;
      DelayOnOff1_2_IN : Bool;
      DelayOnOff1_2_Q : Bool;
      stRefOk : Bool;   // Referans tanımlandı
      stPositionMax : DInt;
      stPositionMin : DInt;
      stConfigEpos : DWord;
      stEposZsw2 : Word;
      stPositive : Bool;   // referans bulma yonu
      stAxisEnabled : Bool;   // OFF1 geldikten sonra setlenir
      Toff1_Instance : TOF_TIME;
      Toff1_IN : Bool;
      Toff1_Q : Bool;
   END_VAR
   VAR_TEMP
      dnPosition : DInt;
      bJog1 : Bool;
      bJog2 : Bool;
      bGoPos : Bool;
      bSetReference : Bool;
      bBusy : Bool;
      bError : Bool;
      bPosDone : Bool;
      rVelocity : Real;
      rOverride : Int;
      nOverride : Int;
      bHomingOff1 : Bool;
      bHomingExecute : Bool;
      bHomingHWLimitActive : Bool;
      bAckError : Bool;
      wAlarm : Word;
      bStandstill : Bool;
   END_VAR
   VAR CONSTANT
      eIDLE : Int := 0;
      eGOPOS_PRE : Int := 1;
      eGOPOS_RUN : Int := 2;
      eREFERENCE_PRE : Int := 3;
      eREFERENCE_RUN : Int := 4;
      eJOG_RUN : Int := 5;
      eJOG_POSITIVE : Int := 6;
      eSUCCESS : Int := 7;
      eERROR : Int := 8;
      eInterrupt : Int := 11;
      eMessage : Int := 12;
      eAxisError : Int := 13;
      eRESET : Int := 14;
   END_VAR
   VAR_TEMP   // added for the SCL form of the ladder/FBD networks
      _w1 : Bool;
      _w2 : Bool;
   END_VAR
BEGIN

REGION Network 2 (SCL): Tanımlamalar
   REGION "TIMER" 
       #IsDoneDelay(IN := #IsDoneDelay_IN,
                    PT := t#400ms,
                    Q => #IsDoneDelay_Q);

       #DelayOnOff1_1(IN := #DelayOnOff1_1_IN,
                      PT := T#300MS,
                      Q => #DelayOnOff1_1_Q);

       #DelayOnOff1_2(IN := #DelayOnOff1_2_IN,
                      PT := T#300MS,
                      Q => #DelayOnOff1_2_Q);

       #Toff1_Instance(IN := #Toff1_IN,
                       PT := t#500ms,
                       Q => #Toff1_Q);
   END_REGION

   REGION "LOCAL DEGISKENLER" 
   (*
       N/M = 1/1 ise 
       PER REVOLUTION = 10000 ise
       BİR TURDA 10mm gider
       Ekrandan gelen pozisyon değerini bin ile çarpılır.
   *)
       #bGoPos := #GoPos;
       #dnPosition := REAL_TO_DINT( #Position * 1000.0 );  // 10000 LU -> 10 mm yapıyor
       #bSetReference := #SetReference;
       #bAckError := #stAxisError AND #AckError;

       #DelayOnOff1_1_IN := NOT #stAxisError AND #Enable;

       #stEnableAxis := #DelayOnOff1_1_Q AND #Enable;

       // #Toff1_IN := #DelayOnOff1_1_Q AND #Enable;
       // #stEnableAxis := #Toff1_Q;

   END_REGION

   REGION "Posizyon Tolerans"

       #stPositionMax := #dnPosition + 4000;
       #stPositionMin := #dnPosition - 4000;

       #IsPosTol := #SINA_POS_Instance_1.ActPosition > #stPositionMin
       AND #SINA_POS_Instance_1.ActPosition < #stPositionMax;

   END_REGION

   REGION "YUZDELIK HIZ HESABI"
       #rVelocity := (#Velocity * 16384.0) / 100.0;
       #stVelocity := REAL_TO_DINT(#rVelocity);  // Hiz bilgisini yukle

   END_REGION

   REGION "JOG HIZ AYARI" 

       #stOverride := #Override;

   END_REGION
END_REGION

REGION Network 3: Baslangic adimi
   // Bos adim
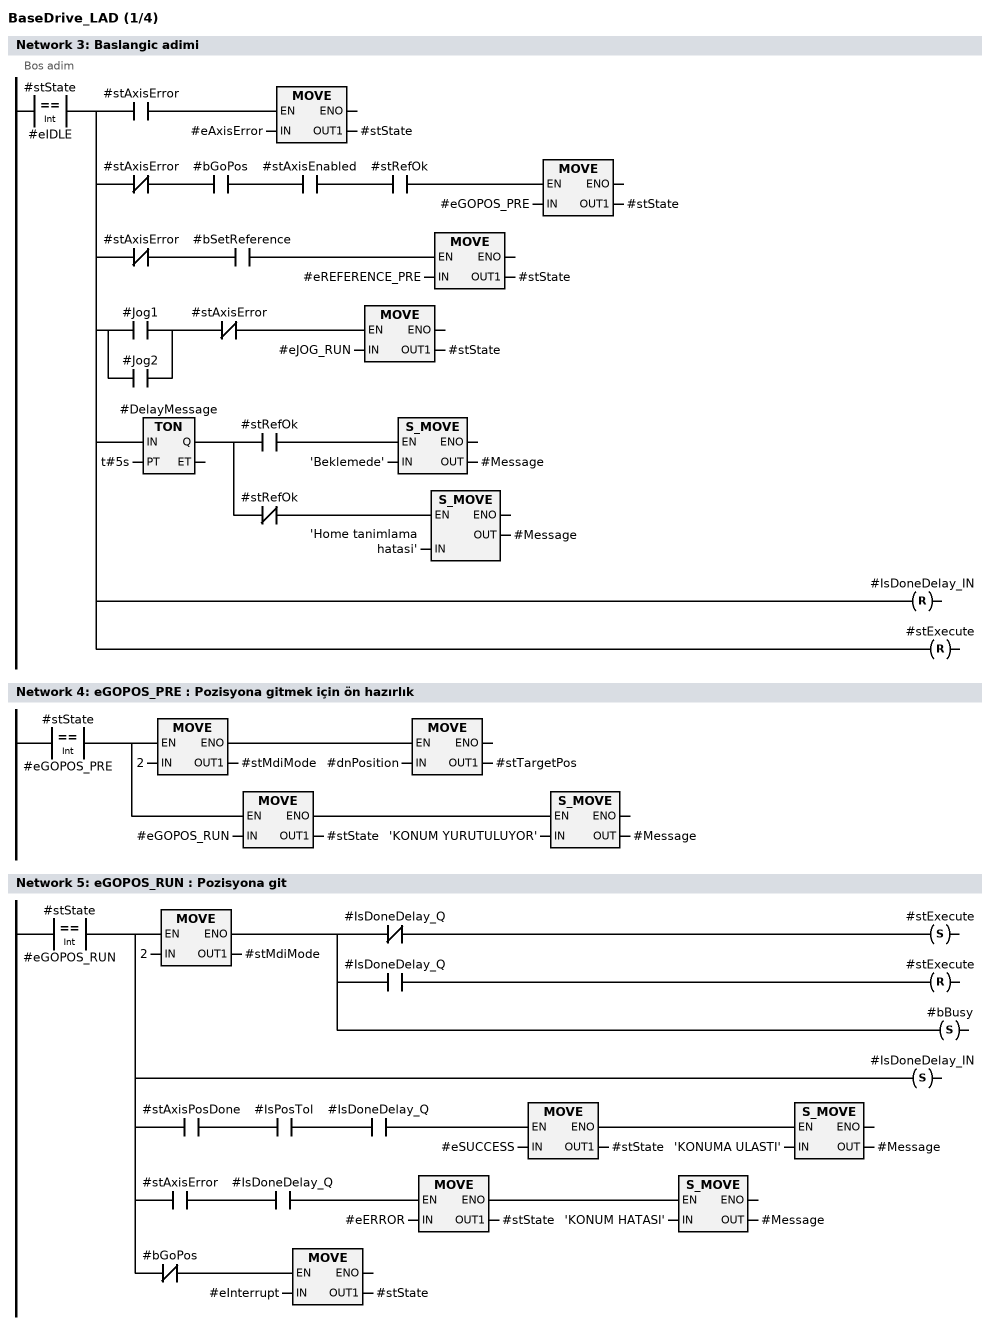
   #_w1 := #stState = #eIDLE;
   IF #_w1 AND #stAxisError THEN #stState := #eAxisError; END_IF;
   IF #_w1 AND NOT #stAxisError AND #bGoPos AND #stAxisEnabled AND #stRefOk THEN
       #stState := #eGOPOS_PRE;
   END_IF;
   IF #_w1 AND NOT #stAxisError AND #bSetReference THEN #stState := #eREFERENCE_PRE; END_IF;
   IF #_w1 AND (#Jog1 OR #Jog2) AND NOT #stAxisError THEN #stState := #eJOG_RUN; END_IF;
   #DelayMessage(IN := #_w1, PT := t#5s);   // TON
   IF #DelayMessage.Q AND #stRefOk THEN #Message := 'Beklemede'; END_IF;
   IF #DelayMessage.Q AND NOT #stRefOk THEN #Message := 'Home tanimlama hatasi'; END_IF;
   IF #_w1 THEN
       #IsDoneDelay_IN := FALSE;
       #stExecute := FALSE;
   END_IF;
END_REGION

REGION Network 4: eGOPOS_PRE : Pozisyona gitmek için ön hazırlık
   RUNG wire#powerrail
      { S7_Templates := "SrcType := Int" } EQ_Contact(in1 := #stState, in2 := #eGOPOS_PRE)
      wire#w1
      Move(in := 2, out1 => #stMdiMode)
      Move(in := #dnPosition, out1 => #stTargetPos)
   END_RUNG
   RUNG wire#w1
      Move(in := #eGOPOS_RUN, out1 => #stState)
      S_Move(in := 'KONUM YURUTULUYOR', out => #Message)
   END_RUNG
   // the same network as SCL:
   IF #stState = #eGOPOS_PRE THEN
       #stMdiMode := 2;
       #stTargetPos := #dnPosition;
   END_IF;
   #_w1 := #stState = #eGOPOS_PRE;
   IF #_w1 THEN
       #stState := #eGOPOS_RUN;
       #Message := 'KONUM YURUTULUYOR';
   END_IF;
END_REGION

REGION Network 5: eGOPOS_RUN : Pozisyona git
   RUNG wire#powerrail
      { S7_Templates := "SrcType := Int" } EQ_Contact(in1 := #stState, in2 := #eGOPOS_RUN)
      wire#w1
      Move(in := 2, out1 => #stMdiMode)
      wire#w2
      I_Contact( #IsDoneDelay_Q )
      S_Coil( #stExecute )
   END_RUNG
   RUNG wire#w2
      Contact( #IsDoneDelay_Q )
      R_Coil( #stExecute )
   END_RUNG
   RUNG wire#w2
      S_Coil( #bBusy )
   END_RUNG
   RUNG wire#w1
      S_Coil( #IsDoneDelay_IN )
   END_RUNG
   RUNG wire#w1
      Contact( #stAxisPosDone )
      Contact( #IsPosTol )
      Contact( #IsDoneDelay_Q )
      Move(in := #eSUCCESS, out1 => #stState)
      S_Move(in := 'KONUMA ULASTI', out => #Message)
   END_RUNG
   RUNG wire#w1
      Contact( #stAxisError )
      Contact( #IsDoneDelay_Q )
      Move(in := #eERROR, out1 => #stState)
      S_Move(in := 'KONUM HATASI', out => #Message)
   END_RUNG
   RUNG wire#w1
      I_Contact( #bGoPos )
      Move(in := #eInterrupt, out1 => #stState)
   END_RUNG
   // the same network as SCL:
   #_w1 := #stState = #eGOPOS_RUN;
   IF #_w1 THEN #stMdiMode := 2; END_IF;
   IF #_w1 AND NOT #IsDoneDelay_Q THEN #stExecute := TRUE; END_IF;
   IF #_w1 AND #IsDoneDelay_Q THEN #stExecute := FALSE; END_IF;
   IF #_w1 THEN
       #bBusy := TRUE;
       #IsDoneDelay_IN := TRUE;
   END_IF;
   IF #_w1 AND #stAxisPosDone AND #IsPosTol AND #IsDoneDelay_Q THEN
       #stState := #eSUCCESS;
       #Message := 'KONUMA ULASTI';
   END_IF;
   IF #_w1 AND #stAxisError AND #IsDoneDelay_Q THEN
       #stState := #eERROR;
       #Message := 'KONUM HATASI';
   END_IF;
   IF #_w1 AND NOT #bGoPos THEN #stState := #eInterrupt; END_IF;
END_REGION

REGION Network 6: Referans belirle
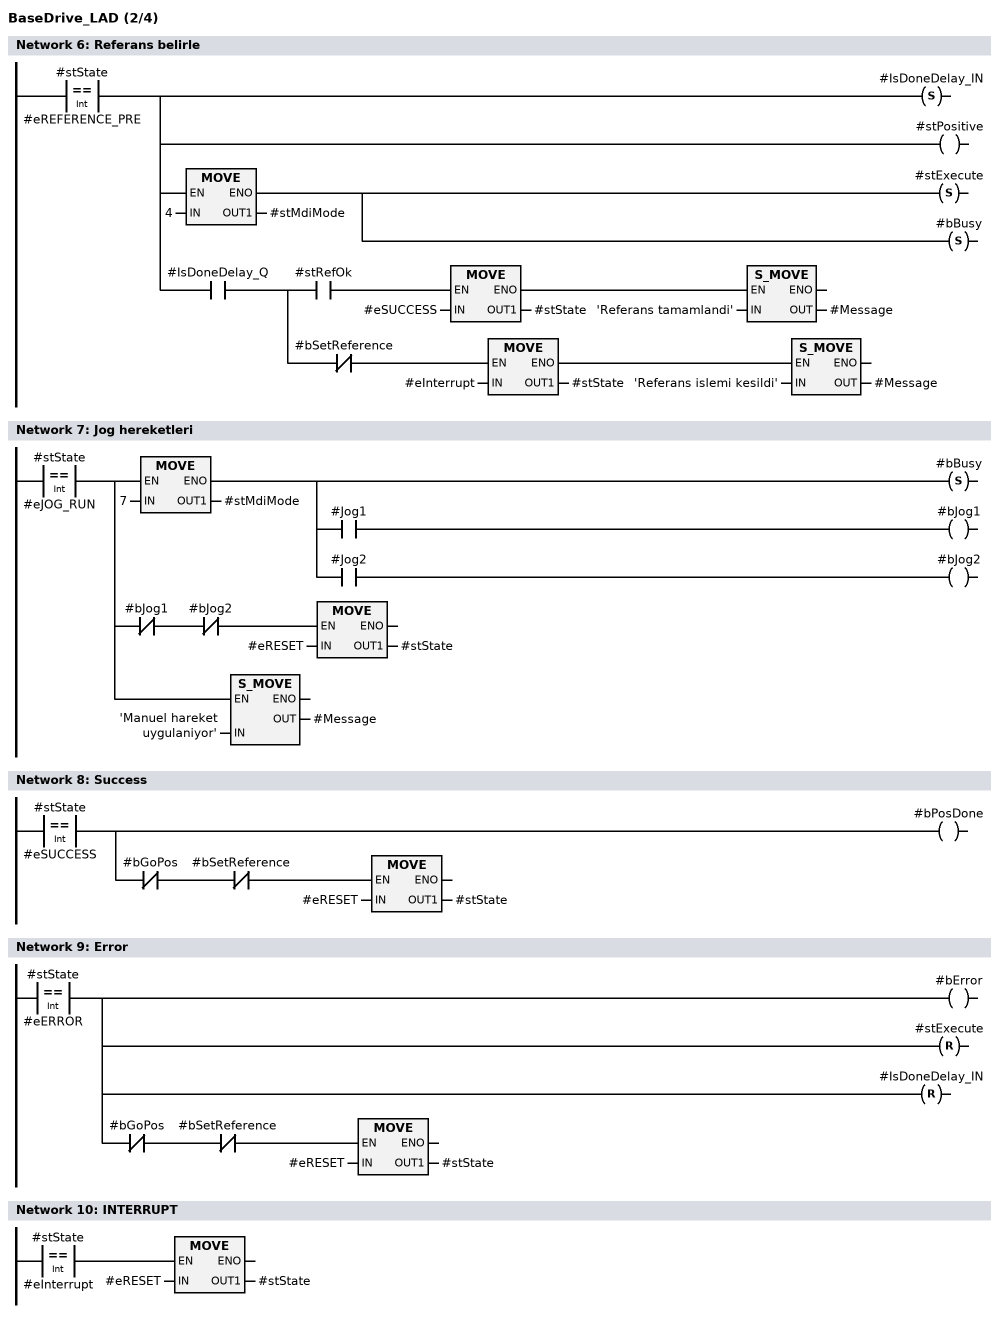
   RUNG wire#powerrail
      { S7_Templates := "SrcType := Int" } EQ_Contact(in1 := #stState, in2 := #eREFERENCE_PRE)
      wire#w1
      S_Coil( #IsDoneDelay_IN )
   END_RUNG
   RUNG wire#w1
      Coil( #stPositive )
   END_RUNG
   RUNG wire#w1
      Move(in := 4, out1 => #stMdiMode)
      wire#w2
      S_Coil( #stExecute )
   END_RUNG
   RUNG wire#w2
      S_Coil( #bBusy )
   END_RUNG
   RUNG wire#w1
      Contact( #IsDoneDelay_Q )
      wire#w3
      Contact( #stRefOk )
      Move(in := #eSUCCESS, out1 => #stState)
      S_Move(in := 'Referans tamamlandi', out => #Message)
   END_RUNG
   RUNG wire#w3
      I_Contact( #bSetReference )
      Move(in := #eInterrupt, out1 => #stState)
      S_Move(in := 'Referans islemi kesildi', out => #Message)
   END_RUNG
   // the same network as SCL:
   #_w1 := #stState = #eREFERENCE_PRE;
   IF #_w1 THEN #IsDoneDelay_IN := TRUE; END_IF;
   #stPositive := #_w1;
   IF #_w1 THEN
       #stMdiMode := 4;
       #stExecute := TRUE;
       #bBusy := TRUE;
   END_IF;
   #_w2 := #_w1 AND #IsDoneDelay_Q;
   IF #_w2 AND #stRefOk THEN
       #stState := #eSUCCESS;
       #Message := 'Referans tamamlandi';
   END_IF;
   IF #_w2 AND NOT #bSetReference THEN
       #stState := #eInterrupt;
       #Message := 'Referans islemi kesildi';
   END_IF;
END_REGION

REGION Network 7: Jog hereketleri
   RUNG wire#powerrail
      { S7_Templates := "SrcType := Int" } EQ_Contact(in1 := #stState, in2 := #eJOG_RUN)
      wire#w1
      Move(in := 7, out1 => #stMdiMode)
      wire#w2
      S_Coil( #bBusy )
   END_RUNG
   RUNG wire#w2
      Contact( #Jog1 )
      Coil( #bJog1 )
   END_RUNG
   RUNG wire#w2
      Contact( #Jog2 )
      Coil( #bJog2 )
   END_RUNG
   RUNG wire#w1
      I_Contact( #bJog1 )
      I_Contact( #bJog2 )
      Move(in := #eRESET, out1 => #stState)
   END_RUNG
   RUNG wire#w1
      S_Move(in := 'Manuel hareket uygulaniyor', out => #Message)
   END_RUNG
   // the same network as SCL:
   #_w1 := #stState = #eJOG_RUN;
   IF #_w1 THEN
       #stMdiMode := 7;
       #bBusy := TRUE;
   END_IF;
   #bJog1 := #_w1 AND #Jog1;
   #bJog2 := #_w1 AND #Jog2;
   IF #_w1 AND NOT #bJog1 AND NOT #bJog2 THEN #stState := #eRESET; END_IF;
   IF #_w1 THEN #Message := 'Manuel hareket uygulaniyor'; END_IF;
END_REGION

REGION Network 8: Success
   RUNG wire#powerrail
      { S7_Templates := "SrcType := Int" } EQ_Contact(in1 := #stState, in2 := #eSUCCESS)
      wire#w1
      Coil( #bPosDone )
   END_RUNG
   RUNG wire#w1
      I_Contact( #bGoPos )
      I_Contact( #bSetReference )
      Move(in := #eRESET, out1 => #stState)
   END_RUNG
   // the same network as SCL:
   #bPosDone := #stState = #eSUCCESS;
   IF #bPosDone AND NOT #bGoPos AND NOT #bSetReference THEN #stState := #eRESET; END_IF;
END_REGION

REGION Network 9: Error
   RUNG wire#powerrail
      { S7_Templates := "SrcType := Int" } EQ_Contact(in1 := #stState, in2 := #eERROR)
      wire#w1
      Coil( #bError )
   END_RUNG
   RUNG wire#w1
      R_Coil( #stExecute )
   END_RUNG
   RUNG wire#w1
      R_Coil( #IsDoneDelay_IN )
   END_RUNG
   RUNG wire#w1
      I_Contact( #bGoPos )
      I_Contact( #bSetReference )
      Move(in := #eRESET, out1 => #stState)
   END_RUNG
   // the same network as SCL:
   #bError := #stState = #eERROR;
   IF #bError THEN
       #stExecute := FALSE;
       #IsDoneDelay_IN := FALSE;
   END_IF;
   IF #bError AND NOT #bGoPos AND NOT #bSetReference THEN #stState := #eRESET; END_IF;
END_REGION

REGION Network 10: INTERRUPT
   RUNG wire#powerrail
      { S7_Templates := "SrcType := Int" } EQ_Contact(in1 := #stState, in2 := #eInterrupt)
      Move(in := #eRESET, out1 => #stState)
   END_RUNG
   // the same network as SCL:
   IF #stState = #eInterrupt THEN #stState := #eRESET; END_IF;
END_REGION

REGION Network 11: RESET
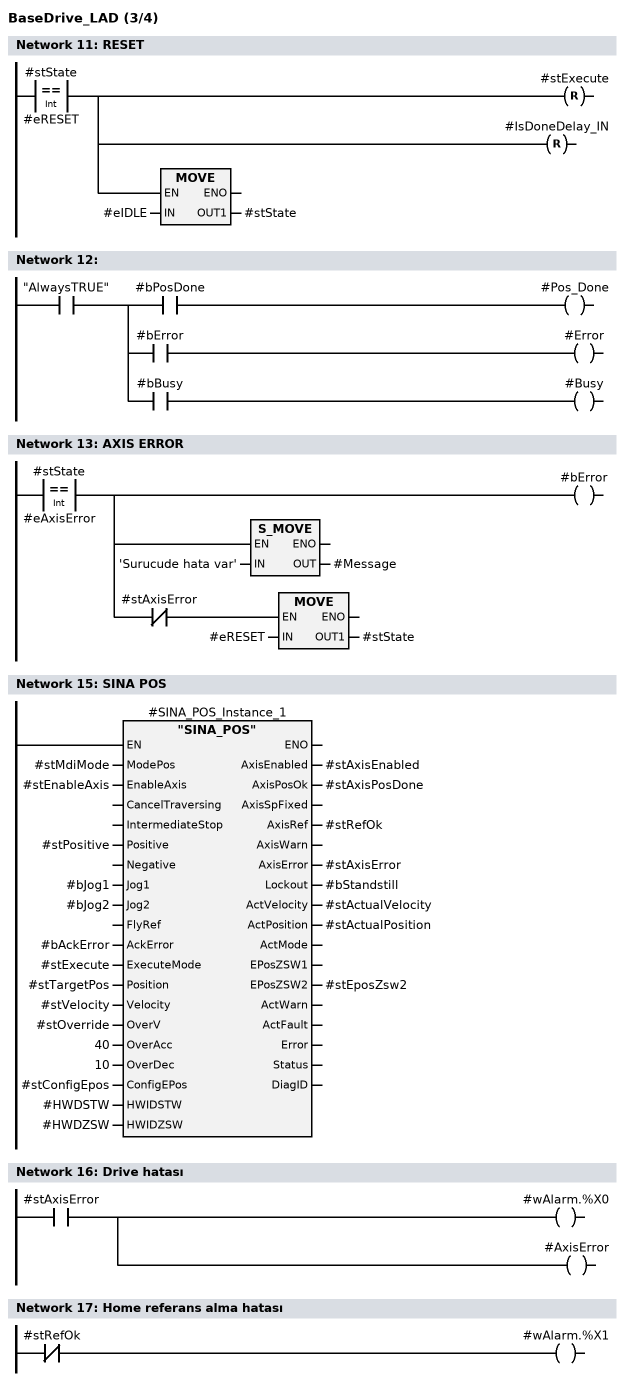
   RUNG wire#powerrail
      { S7_Templates := "SrcType := Int" } EQ_Contact(in1 := #stState, in2 := #eRESET)
      wire#w1
      R_Coil( #stExecute )
   END_RUNG
   RUNG wire#w1
      R_Coil( #IsDoneDelay_IN )
   END_RUNG
   RUNG wire#w1
      Move(in := #eIDLE, out1 => #stState)
   END_RUNG
   // the same network as SCL:
   IF #stState = #eRESET THEN
       #stExecute := FALSE;
       #IsDoneDelay_IN := FALSE;
       #stState := #eIDLE;
   END_IF;
END_REGION

REGION Network 12
   RUNG wire#powerrail
      Contact( "AlwaysTRUE" )
      wire#w1
      Contact( #bPosDone )
      Coil( #Pos_Done )
   END_RUNG
   RUNG wire#w1
      Contact( #bError )
      Coil( #Error )
   END_RUNG
   RUNG wire#w1
      Contact( #bBusy )
      Coil( #Busy )
   END_RUNG
   // the same network as SCL:
   #Pos_Done := "AlwaysTRUE" AND #bPosDone;
   #Error := "AlwaysTRUE" AND #bError;
   #Busy := "AlwaysTRUE" AND #bBusy;
END_REGION

REGION Network 13: AXIS ERROR
   RUNG wire#powerrail
      { S7_Templates := "SrcType := Int" } EQ_Contact(in1 := #stState, in2 := #eAxisError)
      wire#w1
      Coil( #bError )
   END_RUNG
   RUNG wire#w1
      S_Move(in := 'Surucude hata var', out => #Message)
   END_RUNG
   RUNG wire#w1
      I_Contact( #stAxisError )
      Move(in := #eRESET, out1 => #stState)
   END_RUNG
   // the same network as SCL:
   #bError := #stState = #eAxisError;
   IF #bError THEN #Message := 'Surucude hata var'; END_IF;
   IF #bError AND NOT #stAxisError THEN #stState := #eRESET; END_IF;
END_REGION

REGION Network 14 (SCL): Config Epos datasi
   #stConfigEpos.%X0 := TRUE; // default -> OFF2
   #stConfigEpos.%X1 := #Emergency; // default -> OFF3
   #stConfigEpos.%X2 := true; // software limit switch active
   (*
       POS_STW2.2 -> reference cam
       Reference Cam ile calisirken
       sensor bilgisi yukarıdaki bite gönderilecek.

       POS_STW2.2 = #stConfigEpos.%X6 bitidir.
   *)
   #stConfigEpos.%X6 := "Peripheral_Data".IN.ServoHomeSen;
END_REGION

REGION Network 15: SINA POS
   RUNG wire#powerrail
      #SINA_POS_Instance_1(ModePos := #stMdiMode, EnableAxis := #stEnableAxis, CancelTraversing :=, IntermediateStop :=, Positive := #stPositive, Negative :=, Jog1 := #bJog1, Jog2 := #bJog2, FlyRef :=, AckError := #bAckError, ExecuteMode := #stExecute, Position := #stTargetPos, Velocity := #stVelocity, OverV := #stOverride, OverAcc := 40, OverDec := 10, ConfigEPos := #stConfigEpos, HWIDSTW := #HWDSTW, HWIDZSW := #HWDZSW, AxisEnabled => #stAxisEnabled, AxisPosOk => #stAxisPosDone, AxisSpFixed =>, AxisRef => #stRefOk, AxisWarn =>, AxisError => #stAxisError, Lockout => #bStandstill, ActVelocity => #stActualVelocity, ActPosition => #stActualPosition, ActMode =>, EPosZSW1 =>, EPosZSW2 => #stEposZsw2, ActWarn =>, ActFault =>, Error =>, Status =>, DiagID =>)
   END_RUNG
   // the same network as SCL:
   #SINA_POS_Instance_1(ModePos := #stMdiMode,   // "SINA_POS"
                        EnableAxis := #stEnableAxis,
                        Positive := #stPositive,
                        Jog1 := #bJog1,
                        Jog2 := #bJog2,
                        AckError := #bAckError,
                        ExecuteMode := #stExecute,
                        Position := #stTargetPos,
                        Velocity := #stVelocity,
                        OverV := #stOverride,
                        OverAcc := 40,
                        OverDec := 10,
                        ConfigEPos := #stConfigEpos,
                        HWIDSTW := #HWDSTW,
                        HWIDZSW := #HWDZSW,
                        AxisEnabled => #stAxisEnabled,
                        AxisPosOk => #stAxisPosDone,
                        AxisRef => #stRefOk,
                        AxisError => #stAxisError,
                        Lockout => #bStandstill,
                        ActVelocity => #stActualVelocity,
                        ActPosition => #stActualPosition,
                        EPosZSW2 => #stEposZsw2);
END_REGION

REGION Network 16: Drive hatası
   RUNG wire#powerrail
      Contact( #stAxisError )
      wire#w1
      Coil( #wAlarm.%X0 )
   END_RUNG
   RUNG wire#w1
      Coil( #AxisError )
   END_RUNG
   // the same network as SCL:
   #wAlarm.%X0 := #stAxisError;
   #AxisError := #stAxisError;
END_REGION

REGION Network 17: Home referans alma hatası
   RUNG wire#powerrail
      I_Contact( #stRefOk )
      Coil( #wAlarm.%X1 )
   END_RUNG
   // the same network as SCL:
   #wAlarm.%X1 := NOT #stRefOk;
END_REGION

REGION Network 18 (SCL): ACT POSITION
   #ActPosition := DINT_TO_REAL(#stActualPosition) / 1000.0;
END_REGION

REGION Network 19: reference point set
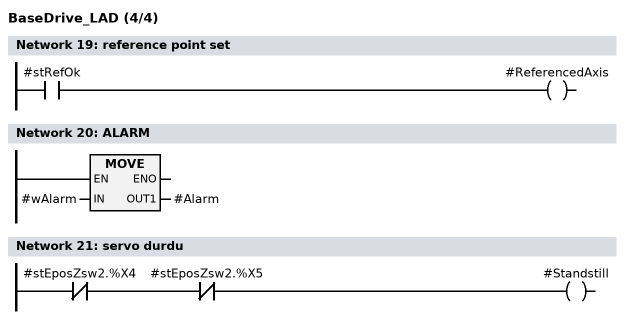
   RUNG wire#powerrail
      Contact( #stRefOk )
      Coil( #ReferencedAxis )
   END_RUNG
   // the same network as SCL:
   #ReferencedAxis := #stRefOk;
END_REGION

REGION Network 20: ALARM
   RUNG wire#powerrail
      Move(in := #wAlarm, out1 => #Alarm)
   END_RUNG
   // the same network as SCL:
   #Alarm := #wAlarm;
END_REGION

REGION Network 21: servo durdu
   RUNG wire#powerrail
      I_Contact( #stEposZsw2.%X4 )
      I_Contact( #stEposZsw2.%X5 )
      Coil( #Standstill )
   END_RUNG
   // the same network as SCL:
   #Standstill := NOT #stEposZsw2.%X4 AND NOT #stEposZsw2.%X5;
END_REGION
END_FUNCTION_BLOCK

FUNCTION_BLOCK "SINA_POS"   // FB284, SCL
TITLE = 'Positioning with SINAMICS and S7'
{ S7_Optimized_Access := 'TRUE' }
AUTHOR : DRVDPS7
FAMILY : DRIVES
NAME : SINA_POS
VERSION : 5.7
// Copyright (C) Siemens AG 2012. All Rights Reserved. Confidential
// -------------------------------------------------------------------------------------- 
// SINA_POS: Positionierung mit dem Antriebsbaustein SINAMICS S120/G120 <-> S7-1200
// ------------------------------------------------------------------------------------- Ersteller: Siemens AG Erlangen A&D MC PM   Datum:  07.07.10        Vers.:2.1
// Änderung:  J.B. Typical Team                       18.12.12              2.2
//     Umsetzung in SCL / TIA 
// Änderung:  J.B. Typical Team                       18.04.13              2.3
//     Bei Betriebsart "Referenzieren - Referenzpunkt setzen"
//     nicht intern setzen sondern Eingang #Execute abfragen als 
//     Startbedingung
// Änderung:  J.B. Typical Team                       29.04.13              2.4
//     1. Off1 möglich bei ungültige Betriebsart
//     2. Referenzpunkt setzen Exceute übernehmen
//     3. Fehlermeldung ausgeben bei Wechel ohne 
//        Beendigung der Betriebsart 
//     4. "Q" an den Ausgänge entfernen
//     5. Neuer Ausgang PwrInhibit
//      
// Änderung:  J.B. Typical Team                       14.05.13              2.5
//     Fehlerbehebung und Defaultwerte ändern
// Änderung:  J.B. Typical Team                       28.06.13              2.6
//     HW-Zugriffsermittlung über LOG2MOD
// Änderung:  J.B. Typical Team                       18.07.13              2.7
//     HW-Zugriffsermittlung über zwei HW-Eingänge
// Änderung:  J.B. Typical Team                       18.09.13              2.8
//     Konvertierungsfehler behoben
// Änderung:  J.B. Typical Team                       25.09.13              2.9
//     Bei Betriebswechsel von 3 nach 6 darf MidStart nicht sitzen
// Änderung:  J.B. Typical Team                       31.03.14              3.0
//     In der Betriebsart 1-3 und 6 darf MidTrTyp nicht sitzen
// Änderung:  J.B. Typical Team                       25.06.14              3.1
//     Das Quittierbit "AckFlt" immer durchreichen
// Änderung:  J.B. Typical Team                       30.07.14              4.0
//     Festlegung auf einheitlicher neuer Version 4.0
// Änderung:  J.B. Typical Team                       07.11.14              4.1
//     Fehlerbehebung falsche Zuweisung von Off1 bei Mode 4
//     und Mode 8(DriveLib V4 - RQ 346046)
// Änderung:  F.G. Typical Team                       16.04.15              4.2
//     Anzahl der Zyklen die auf die Rückmeldung fliegendes Ref.
//     gewartet wird verdoppelt (siRetryMax = 10)  (DriveLib V4 - RQ 367986)
// Änderung:  F.G. Typical Team                       15.09.15              4.3
//     Anzahl der Zyklen die auf die Rückmeldung fliegendes Ref.
//     gewartet noch einmal um 5 erhöht (siRetryMax = 15)  (DriveLib V4 - RQ 367986)
// Änderung:  F.G. Typical Team                       15.09.15              4.4
//     Abfrage des richtigen Bits im EPosZSW1 (Zeile 1394)es muss das Bit12 
//     und nicht das Bit 11 abgefragt werden  (DriveLib V4 - RQ 367986)
// Änderung:  F.G. Typical Team                       03.12.15              4.5
//     1. Ein-/Ausgänge an Programmierleitfaden für TIA-Portal angepasst
//        Zusätzlicher Eingang um alle Bits in den STWs zu bedienen
//     2. Warnung durch Initialisierung elimininiert
// Änderung:  F.G. Typical Team                       13.09.16              4.6
//     Ausgabewerte am Ausgang "Status" angepasst 
// 
// Änderung:  G.F. Typical Team                       11.01.17              5.0
//     - Festlegung auf einheitlicher neuer Version 5.0 
// 
// Änderung:  G.F. Typical Team                       13.07.17              5.1
//     - Zuordnung der Bits von ConfigPos korrigiert 
// 
// Änderung:  G.F. Typical Team                       12.01.18              5.2
//     - RQ2637983 sxSendBuf.EPosSTW2.%X1 in Mode 7 und 8 rücksetzen 
// Änderung:  G.F. Typical Team                       20.07.18              5.3
//     - ZSW1.13 als Ausgang zur Verfügung gestellt (wegen FW - Änderung)
// Änderung:  G.F. Typical Team                       18.10.18              5.4
//     - RQ 824321 Zähler für fliegendes Referenzieren zurücksetzen
// Änderung:  G.F. Typical Team                       08.02.19              5.5
//     - Version wegen Änderungen in älteren Lib-Versionen 
// Änderung:  G.F. Typical Team                       08.02.19              5.6
//     - RQ 3901129 Fehler Flankenauswertung Eingang ExecuteMode behoben Bibliothek V7
// Änderung:  G.F. Typical Team                       17.05.19              5.7
//     - RQ 4094299 Fehler Referenzfahrt wird nicht gestartet behoben Bibliothek V7
// Funktion: Positionierung mit dem Antriebsbaustein SINAMICS S120/G120 <-> S7-1200
// ********************************************************************************************************************************************************
// ************************************************************************FB283***************************************************************************
// ********************************************************************************************************************************************************
// Copyright (C) Siemens AG 2012. All Rights Reserved. Confidential
// -------------------------------------------------------------------------------------- 
// SINA_POS: Positionierung mit dem Antriebsbaustein SINAMICS S120/G120 <-> S7-1200
// ------------------------------------------------------------------------------------- Ersteller: Siemens AG Erlangen A&D MC PM   Datum:  07.07.10        Vers.:2.1
// Änderung:  J.B. Typical Team                       18.12.12              2.2
//     Umsetzung in SCL / TIA 
// Änderung:  J.B. Typical Team                       18.04.13              2.3
//     Bei Betriebsart "Referenzieren - Referenzpunkt setzen"
//     nicht intern setzen sondern Eingang #Execute abfragen als 
//     Startbedingung
// Änderung:  J.B. Typical Team                       29.04.13              2.4
//     1. Off1 möglich bei ungültige Betriebsart
//     2. Referenzpunkt setzen Exceute übernehmen
//     3. Fehlermeldung ausgeben bei Wechel ohne 
//        Beendigung der Betriebsart 
//     4. "Q" an den Ausgänge entfernen
//     5. Neuer Ausgang PwrInhibit
//      
// Änderung:  J.B. Typical Team                       14.05.13              2.5
//     Fehlerbehebung und Defaultwerte ändern
// Änderung:  J.B. Typical Team                       28.06.13              2.6
//     HW-Zugriffsermittlung über LOG2MOD
// Änderung:  J.B. Typical Team                       18.07.13              2.7
//     HW-Zugriffsermittlung über zwei HW-Eingänge
// Änderung:  J.B. Typical Team                       18.09.13              2.8
//     Konvertierungsfehler behoben
// Änderung:  J.B. Typical Team                       25.09.13              2.9
//     Bei Betriebswechsel von 3 nach 6 darf MidStart nicht sitzen
// Änderung:  J.B. Typical Team                       31.03.14              3.0
//     In der Betriebsart 1-3 und 6 darf MidTrTyp nicht sitzen
// Änderung:  J.B. Typical Team                       25.06.14              3.1
//     Das Quittierbit "AckFlt" immer durchreichen
// Änderung:  J.B. Typical Team                       30.07.14              4.0
//     Festlegung auf einheitlicher neuer Version 4.0
// Änderung:  J.B. Typical Team                       07.11.14              4.1
//     Fehlerbehebung falsche Zuweisung von Off1 bei Mode 4
//     und Mode 8(DriveLib V4 - RQ 346046)
// Änderung:  F.G. Typical Team                       16.04.15              4.2
//     Anzahl der Zyklen die auf die Rückmeldung fliegendes Ref.
//     gewartet wird verdoppelt (siRetryMax = 10)  (DriveLib V4 - RQ 367986)
// Änderung:  F.G. Typical Team                       15.09.15              4.3
//     Anzahl der Zyklen die auf die Rückmeldung fliegendes Ref.
//     gewartet noch einmal um 5 erhöht (siRetryMax = 15)  (DriveLib V4 - RQ 367986)
// Änderung:  F.G. Typical Team                       15.09.15              4.4
//     Abfrage des richtigen Bits im EPosZSW1 (Zeile 1394)es muss das Bit12 
//     und nicht das Bit 11 abgefragt werden  (DriveLib V4 - RQ 367986)
// Änderung:  F.G. Typical Team                       03.12.15              4.5
//     1. Ein-/Ausgänge an Programmierleitfaden für TIA-Portal angepasst
//        Zusätzlicher Eingang um alle Bits in den STWs zu bedienen
//     2. Warnung durch Initialisierung elimininiert
// Änderung:  F.G. Typical Team                       13.09.16              4.6
//     Ausgabewerte am Ausgang "Status" angepasst 
// 
// Änderung:  G.F. Typical Team                       11.01.17              5.0
//     - Festlegung auf einheitlicher neuer Version 5.0 
// 
// Änderung:  G.F. Typical Team                       13.07.17              5.1
//     - Zuordnung der Bits von ConfigPos korrigiert 
// 
// Änderung:  G.F. Typical Team                       12.01.18              5.2
//     - RQ2637983 sxSendBuf.EPosSTW2.%X1 in Mode 7 und 8 rücksetzen 
// Änderung:  G.F. Typical Team                       20.07.18              5.3
//     - ZSW1.13 als Ausgang zur Verfügung gestellt (wegen FW - Änderung)
// Änderung:  G.F. Typical Team                       18.10.18              5.4
//     - RQ 824321 Zähler für fliegendes Referenzieren zurücksetzen
// Änderung:  G.F. Typical Team                       08.02.19              5.5
//     - Version wegen Änderungen in älteren Lib-Versionen 
// Änderung:  G.F. Typical Team                       08.02.19              5.6
//     - RQ 3901129 Fehler Flankenauswertung Eingang ExecuteMode behoben Bibliothek V7
// Funktion: Positionierung mit dem Antriebsbaustein SINAMICS S120/G120 <-> S7-1200
// ********************************************************************************************************************************************************
// ************************************************************************FB283***************************************************************************
// ********************************************************************************************************************************************************
   VAR_INPUT
      ModePos : Int := 0;   // Settings of the mode / Auswahl EPos Betriebsart (0= keine; 1,2,3 = MDI; 4,5 = Referenzieren; 6= Verfarhsätze; 7,8 = Tippen)
      EnableAxis : Bool := 0;   // 1 = Enable the drive / 0-->1 = Einschalten des Antriebs (OFF1 = 0-->1)
      CancelTraversing : Bool := 1;   // 0 = Reject active traverse task / 0 = Abruch der laufenden Verfahrbewegung (1=kein Abbruch)
      IntermediateStop : Bool := 1;   // 0 = Intermediate STOP of traverse command / 0 = Zwischenhalt der laufenden Verfahrbewegung (1= kein Zwischenhalt)
      Positive : Bool := 0;   // 1 = Direction positive / 1 = Positive Verfahrrichtung
      Negative : Bool := 0;   // 1 = Direction negative / 1 = Negative Verfahrrichtung
      Jog1 : Bool := 0;   // 1 = Use jog 1 (direction / speed) / 1 = Tippen Sollwert 1 auswählen
      Jog2 : Bool := 0;   // 1 = Use jog 2 (direction / speed) / 1 = Tippen Sollwert 2 auswählen
      FlyRef : Bool := 0;   // 1 = Start flying reference function / 1 = Aktivierung Fliegendes Referenzieren (nicht möglich bei ModePos = 4, 5)
      AckError : Bool := 0;   // 1 = Acknowledge of errors / 1 = Achs / EPos Fehlerquittierung anwählen
      ExecuteMode : Bool := 0;   // 0-->1 = Start the mode / 0-->1 = Starten der mit ModePos gewählten Betriebsart
      Position : DInt := 0;   // Position of the MDI mode or setting of traversing block / Positionssollwert [LU] für Direkt Sollwert vorgabe (MDI)
      Velocity : DInt := 0;   // MDI velocity / MDI Geschwindigkeit [1000*LU / min]
      OverV : Int := 100;   // Override of velocity in [%] --> 4000h=100% / Geschwindigkeit Skalierung (Alle Betriebsarten 4000h = 100%))
      OverAcc : Int := 100;   // Override of acceleration in [%] --> 4000h=100% / MDI Beschleunigung (4000h = 100%)
      OverDec : Int := 100;   // Override of deceleration in [%] --> 4000h=100% / MDI Verzögerung (4000h = 100%)
      ConfigEPos : DWord := 16#0000_0003;   // binary programmed input to control all functions in the telegram without its own function block input / Binärcodierter Eingang zur Ansteuerung aller nicht als Bausteineingang verfügbaren Steuerbits
      HWIDSTW : Hw_Io := 0;   // Hardware Identifer set point slot / Hardware Identifer des Sollwert Slots
      HWIDZSW : Hw_Io := 0;   // Hardware Identifer actual value slot / Hardware Identifer des Istwert Slots
   END_VAR
   VAR_OUTPUT
      AxisEnabled : Bool := 0;   // 1= Axis in operation / 1= EPos Achse ist in Betrieb
      AxisPosOk : Bool := 0;   // 1= Position setpoint reached / 1= EPos Achsposition erreicht
      AxisSpFixed : Bool := 0;   // 1= Setpoint fixed (Attention: Dependence on SINAMICS firmware) / 1= Sollwert steht (Achtung: Abhängigkeit von SINAMICS Firmware)
      AxisRef : Bool := 0;   // 1= Reference point set / 1= EPos Achse referenziert
      AxisWarn : Bool := 0;   // 1= Axis alarm / warning present / 1= Antriebswarnung aktiv
      AxisError : Bool := 0;   // 1= Axis fault present / 1= Antriebs / EPos Fehler vorhanden
      Lockout : Bool := 0;   // 1= Axis in lockout state / 1= Einschaltsperre aktiv
      ActVelocity : DInt := 0;   // Actual drive speed (has to be normed with p2000 --> 40000000h = 100%) / Aktuelle Geschwindigkeit (40000000h = 100% von p2000 in [rpm])
      ActPosition : DInt := 0;   // Actual position in [LU] / Aktuelle Position in LU
      ActMode : Int := 0;   // Active EPos mode / Aktuellle Betriebsart
      EPosZSW1 : Word := 0;   // Status of EPOS ZSW1
      EPosZSW2 : Word := 0;   // Status of EPOS ZSW2
      ActWarn : Word := 0;   // Actual number of warning / Aktuelle Warnung
      ActFault : Word := 0;   // Actual number of error / Aktuelle Störung
      Error : Bool := 0;   // 1 = Error (FB and Infeed) / Fehler (Antrieb und / oder Funktionsbaustein)
      Status : Word := 0;   // Status output (7002 = FB in operation; 8xxx = error description - read the manual) / Statusausgabe (7002 = FB in Betrieb; 8xxx = Feherbeschreibung siehe Doku)
      DiagID : Word := 0;   // Error codes of the cyclic system funtion blocks DPWR / DPRD_DAT / Fehlercode der zyklischen Systemfunktionen DPWR / DPRD_DAT
   END_VAR
   VAR
      sbOff1Edge : Bool := 0;   // Positive edge of starting or stopping the device
      sbOff1 : Bool := 0;   // Starting or stopping the device
      sbExecuteEdge : Bool := 0;   // Positive edge of activate traversing block
      sbExecute : Bool := 0;   // Activate traversing block
      sbRefTypEdge : Bool := 0;   // Positive edge of referencing type "flying reference"
      sbRefTyp : Bool := 0;   // Referencing type "flying reference"
      sbMdiStart : Bool := 0;   // Direct setpoint input / MDI - start
      sbMdiStartEdge : Bool := 0;   // Positive edge of direct setpoint input / MDI - start
      sbRefStart : Bool := 0;   // Referencing start
      sbJogInc : Bool := 0;   // Jogging incremental
      sbReady : Bool := 0;   // Ready to power up / to start
      sbIOp : Bool := 0;   // Ready to operate
      sbAccel : Bool := 0;   // Axis accelerating
      sbDecel : Bool := 0;   // Axis decelerating
      sbAlarm : Bool := 0;   // Alarm / Warnung present
      sbFault : Bool := 0;   // Fault present
      sbFWD : Bool := 0;   // Axis drives forwards
      sbBWD : Bool := 0;   // Axis drives backwards
      sbBusy : Bool := 0;   // Mode of operation is explained
      swStatus : Word := 16#0000;   // Mode of operation disturbance
      swEPosZSW1 : Word := 16#0000;   // Status of EPOS ZSW1 / EPos Zustandswort 1
      swEPosZSW2 : Word := 16#0000;   // Status of EPOS ZSW2 / EPos Zustandswort 2
      siExecuteCyc : Int := 0;   // Counter of runcycle of active traversing block
      siRefTypCyc : Int := 0;   // Counter of runcycle of referencing type "flying reference"
      siJogIncCyc : Int := 0;   // Counter of runcycle of jogging incremental
      siMdiStartCyc : Int := 0;   // Counter of runcycle of direct setpoint input / MDI - start
      siRefActRetry : Int := 0;   // Counter of retry of reference point approach active
      siModePos : Int := 0;   // Setting of mode
      siModePosMax : Int := 8;   // Max. count of mode
      siCycWait : Int := 5;   // Counter of cycle of waiting
      siRetryMax : Int := 30;   // Max. count of cycles of retry
      sbModePos : Bool := 0;   // Mode of setting okay
      sxSendBuf : Struct   // send buffer of telegram for sending data to the drive
         STW1 : Word := WORD#16#0000;   // STW1sxSTW1 : STRUCT Jog1 : BOOL:=0; // ST-Wort-1 Bit 08 --> 1 = Jogging - signal source 1 Jog2 : BOOL:=0; // ST-Wort-1 Bit 09 --> 1 = Jogging - signal source 2 LB : BOOL:=1; // Allways // ST-Wort-1 Bit 10 --> 1 = Life bit RefStart : BOOL:=0; // ST-Wort-1 Bit 11 --> 1 = Referencing start / stop Bit12 : BOOL:=0; // ST-Wort-1 Bit 12 --> 1 = Reserve Bit13 : BOOL:=0; // ST-Wort-1 Bit 13 --> 1 = Externer Satzwechsel Bit14 : BOOL:=0; // ST-Wort-1 Bit 14 --> 1 = Reserve Bit15 : BOOL:=0; // ST-Wort-1 Bit 15 --> 1 = Reserve Off1 : BOOL:=0; // ST-Wort-1 Bit 00 --> 1 = OFF1/ON (flanks acceptance) Off2 : BOOL:=1; // Allways // ST-Wort-1 Bit 01 --> 1 = OFF2/ON (enable possible) Off3 : BOOL:=1; // Allways // ST-Wort-1 Bit 02 --> 1 = OFF3/ON (enable possible) Enc : BOOL:=1; // Allways // ST-Wort-1 Bit 03 --> 1 = Enable controller RejTrvTsk : BOOL:=0; // ST-Wort-1 Bit 04 --> 1 = Traversing block and MDI - reject task IntMStop : BOOL:=0; // ST-Wort-1 Bit 05 --> 1 = Traversing block and MDI - intermediate - STOP TrvStart : BOOL:=0; // ST-Wort-1 Bit 06 --> 1 = Traversing start - direct setpoint input / MDI - transfer edge AckFault : BOOL:=0; // ST-Wort-1 Bit 07 --> 1 = Acknowledge fault END_STRUCT;
         EPosSTW1 : Word := WORD#16#0000;   // EPOSSTW1sxEPosSTW1 : STRUCT MdiTyp : BOOL:=0; // EPOS-Wort-1 Bit 08 --> 1 = Direct setpoint input / MDI - positioning type MdiPos : BOOL:=0; // EPOS-Wort-1 BIT 09 --> 1 = Direct setpoint input / MDI - positive direction MdiNeg : BOOL:=0; // EPOS-Wort-1 BIT 10 --> 1 = Direct setpoint input / MDI - negative direction Bit11 : BOOL:=0; // EPOS-Wort-1 BIT 11 --> 1 = Reserve MdiTrTyp : BOOL:=0; // EPOS-Wort-1 BIT 12 --> 1 = Direct setpoint input / MDI - transfer type Bit13 : BOOL:=0; // EPOS-Wort-1 BIT 13 --> 1 = Reserve MdiSetup : BOOL:=0; // EPOS-Wort-1 BIT 14 --> 1 = Direct setpoint input / MDI - setup selection MdiStart : BOOL:=0; // EPOS-Wort-1 BIT 15 --> 1 = Direct setpoint input / MDI - start TrvBit0 : BOOL:=0; // EPOS-Wort-1 BIT 00 --> 1 = Traversing block - block selection bit 0 TrvBit1 : BOOL:=0; // EPOS-Wort-1 BIT 01 --> 1 = Traversing block - block selection bit 1 TrvBit2 : BOOL:=0; // EPOS-Wort-1 BIT 02 --> 1 = Traversing block - block selection bit 2 TrvBit3 : BOOL:=0; // EPOS-Wort-1 BIT 03 --> 1 = Traversing block - block selection bit 3 TrvBit4 : BOOL:=0; // EPOS-Wort-1 BIT 04 --> 1 = Traversing block - block selection bit 4 TrvBit5 : BOOL:=0; // EPOS-Wort-1 Bit 05 --> 1 = Traversing block - block selection bit 5 Bit06 : BOOL:=0; // EPOS-Wort-1 Bit 06 --> 1 = Reserve Bit07 : BOOL:=0; // EPOS-Wort-1 Bit 07 --> 1 = Reserve END_STRUCT;
         EPosSTW2 : Word := WORD#16#0000;   // EPOSSTW2sxEPosSTW2 : STRUCT RefTyp : BOOL:=0; // EPOS-Wort-2 Bit 08 --> 1 = Referencing type RefStDi : BOOL:=0; // EPOS-Wort-2 Bit 09 --> 1 = Homing start direction RefInpS : BOOL:=0; // EPOS-Wort-2 Bit 10 --> 1 = Referencing passive - input selection RefEdge : BOOL:=0; // EPOS-Wort-2 Bit 11 --> 1 = Referencing passive - edge evaluation Bit12 : BOOL:=0; // EPOS-Wort-2 Bit 12 --> 1 = Reserve Bit13 : BOOL:=0; // EPOS-Wort-2 Bit 13 --> 1 = Reserve SftLimAct : BOOL:=0; // EPOS-Wort-2 Bit 14 --> 1 = Software limit switch activation StpCamAct : BOOL:=0; // EPOS-Wort-2 Bit 15 --> 1 = Stop output cam activation TrkMode : BOOL:=0; // EPOS-Wort-2 Bit 00 --> 1 = Tracking mode active SetRefPt : BOOL:=0; // EPOS-Wort-2 Bit 01 --> 1 = Set reference point ActRefCam : BOOL:=0; // EPOS-Wort-2 Bit 02 --> 1 = Reference cam active Bit03 : BOOL:=0; // EPOS-Wort-2 Bit 03 --> 1 = Reserve Bit04 : BOOL:=0; // EPOS-Wort-2 Bit 04 --> 1 = Reserve JogInc : BOOL:=0; // EPOS-Wort-2 Bit 05 --> 1 = Jogging - jogging incremental Bit06 : BOOL:=0; // EPOS-Wort-2 Bit 06 --> 1 = Reserve Bit07 : BOOL:=0; // EPOS-Wort-2 Bit 07 --> 1 = Reserve END_STRUCT;
         STW2 : Word := WORD#16#0000;   // STW2sxSTW2 : STRUCT TrvFixStp : BOOL:=0; // ST-Wort-2 Bit 08 --> 1 = Travel fixed STOP GlbTrgCom : BOOL:=0; // ST-Wort-2 Bit 09 --> 1 = Global trigger command Bit10 : BOOL:=0; // ST-Wort-2 Bit 10 --> 1 = Reserve MotSwOver : BOOL:=0; // ST-Wort-2 Bit 11 --> 1 = Motor switch over finished MsZykBit0 : BOOL:=0; // ST-Wort-2 Bit 12 --> 1 = Master life bit 0 MsZykBit1 : BOOL:=0; // ST-Wort-2 Bit 13 --> 1 = Master life bit 1 MsZykBit2 : BOOL:=0; // ST-Wort-2 Bit 14 --> 1 = Master life bit 2 MsZykBit3 : BOOL:=0; // ST-Wort-2 Bit 15 --> 1 = Master life bit 3 DDSBit0 : BOOL:=0; // ST-Wort-2 Bit 00 --> 1 = Drive data set bit 0 DDSBit1 : BOOL:=0; // ST-Wort-2 Bit 01 --> 1 = Drive data set bit 1 DDSBit2 : BOOL:=0; // ST-Wort-2 Bit 02 --> 1 = Drive data set bit 2 DDSBit3 : BOOL:=0; // ST-Wort-2 Bit 03 --> 1 = Drive data set bit 3 DDSBit4 : BOOL:=0; // ST-Wort-2 Bit 04 --> 1 = Drive data set bit 4 GlbStart : BOOL:=0; // ST-Wort-2 Bit 05 --> 1 = Global start ResIComp : BOOL:=0; // ST-Wort-2 Bit 06 --> 1 = Reset I-component of speed controller ActPrkAxis : BOOL:=0; // ST-Wort-2 Bit 07 --> 1 = Activate parking axis END_STRUCT;
         OverrideV : Word := WORD#16#0000;   // Velocity override
         Position : DWord := DWORD#16#0000_0000;   // Setpoint of position
         Velocity : DWord := DWORD#16#0000_0000;   // Setpoint of velocity
         OverrideA : Word := WORD#16#0000;   // Accelerating override
         OverrideD : Word := WORD#16#0000;   // Decelerating override
         Reserve : Word := WORD#16#0000;   // Reserve
      END_STRUCT;
      sxRecvBuf : Struct   // receive buffer of telegram for receiving data from the drive
         ZSW1 : Word := WORD#16#0000;   // ZSW1sxZSW1 : STRUCT NoFlwErr : BOOL:=0; // ZSW-Wort-1 Bit 08 --> 1 = Following error in tolerance LbCr : BOOL:=0; // ZSW-Wort-1 Bit 09 --> 1 = Lifebit control request TargPos : BOOL:=0; // ZSW-Wort-1 Bit 10 --> 1 = Target position reached RefPSet : BOOL:=0; // ZSW-Wort-1 Bit 11 --> 1 = Reference point set TrvTskAck : BOOL:=0; // ZSW-Wort-1 Bit 12 --> 1 = Traversing task acknowledge StndStill : BOOL:=0; // ZSW-Wort-1 Bit 13 --> 1 = [n_ist] < Drehzahlsollwert 3 Accel : BOOL:=0; // ZSW-Wort-1 Bit 14 --> 1 = Axis accelerating Decel : BOOL:=0; // ZSW-Wort-1 Bit 15 --> 1 = Axis decelerating RTS : BOOL:=0; // ZSW-Wort-1 Bit 00 --> 1 = Ready to power up / to start RDY : BOOL:=0; // ZSW-Wort-1 Bit 01 --> 1 = Ready to operate IOp : BOOL:=0; // ZSW-Wort-1 Bit 02 --> 1 = In operation (operation enabled) Fault : BOOL:=0; // ZSW-Wort-1 Bit 03 --> 1 = Fault present NoOff2Act : BOOL:=0; // ZSW-Wort-1 Bit 04 --> 1 = OFF2 inactive NoOff3Act : BOOL:=0; // ZSW-Wort-1 Bit 05 --> 1 = OFF3 inactive PowInhbt : BOOL:=0; // ZSW-Wort-1 Bit 06 --> 1 = Power ON inhibit active Alarm : BOOL:=0; // ZSW-Wort-1 Bit 07 --> 1 = Alarm / Warning present END_STRUCT;
         EPosZSW1 : Word := WORD#16#0000;   // EPOSZSW1sxEPosZSW1 : STRUCT StpCamMinAct : BOOL:=0; // EPOS-Wort-1 Bit 08 --> 1 = STOP cam minus active StpCamPlsAct : BOOL:=0; // EPOS-Wort-1 Bit 09 --> 1 = STOP cam plus active JogAct : BOOL:=0; // EPOS-Wort-1 Bit 10 --> 1 = Jogging active RefAct : BOOL:=0; // EPOS-Wort-1 Bit 11 --> 1 = Reference point approach active FlyRefAct : BOOL:=0; // EPOS-Wort-1 Bit 12 --> 1 = Flying referencing active TrvBlAct : BOOL:=0; // EPOS-Wort-1 Bit 13 --> 1 = Traversing block active MdiStupAct : BOOL:=0; // EPOS-Wort-1 Bit 14 --> 1 = MDI setup active MdiPosAct : BOOL:=0; // EPOS-Wort-1 Bit 15 --> 1 = MDI positing active ActTrvBit0 : BOOL:=0; // EPOS-Wort-1 BIT 00 --> 1 = Active traversing block bit 0 ActTrvBit1 : BOOL:=0; // EPOS-Wort-1 Bit 01 --> 1 = Active traversing block bit 1 ActTrvBit2 : BOOL:=0; // EPOS-Wort-1 Bit 02 --> 1 = Active traversing block bit 2 ActTrvBit3 : BOOL:=0; // EPOS-Wort-1 Bit 03 --> 1 = Active traversing block bit 3 ActTrvBit4 : BOOL:=0; // EPOS-Wort-1 Bit 04 --> 1 = Active traversing block bit 4 ActTrvBit5 : BOOL:=0; // EPOS-Wort-1 Bit 05 --> 1 = Active traversing block bit 5 Bit06 : BOOL:=0; // EPOS-Wort-1 Bit 06 --> 1 = Reserve Bit07 : BOOL:=0; // EPOS-Wort-1 Bit 07 --> 1 = Reserve END_STRUCT;
         EPosZSW2 : Word := WORD#16#0000;   // EPOSZSW2sxEPosZSW2 : STRUCT PosSmCam1 : BOOL:=0; // EPOS-Wort-2 Bit 08 --> 1 = Position actual value <= cam position 1 PosSmCam2 : BOOL:=0; // EPOS-Wort-2 Bit 09 --> 1 = Position actual value <= cam position 2 TrvOut1 : BOOL:=0; // EPOS-Wort-2 Bit 10 --> 1 = Direct output 1 via traversing block TrvOut2 : BOOL:=0; // EPOS-Wort-2 Bit 11 --> 1 = Direct output 2 via traversing block FxStpRd : BOOL:=0; // EPOS-Wort-2 Bit 12 --> 1 = Fixed STOP reached FxStpTrRd : BOOL:=0; // EPOS-Wort-2 Bit 13 --> 1 = Fixed STOP clamping torque reached TrvFxStpAct : BOOL:=0; // EPOS-Wort-2 Bit 14 --> 1 = Traversing fixed STOP active CmdAct : BOOL:=0; // EPOS-Wort-2 Bit 15 --> 1 = Traversing command active TrkModeAct : BOOL:=0; // EPOS-Wort-2 Bit 00 --> 1 = Tracking mode active VeloLimAct : BOOL:=0; // EPOS-Wort-2 Bit 01 --> 1 = Velocity limit active SetPStat : BOOL:=0; // EPOS-Wort-2 Bit 02 --> 1 = Setpoint static PrnMrkOut : BOOL:=0; // EPOS-Wort-2 Bit 03 --> 1 = Printmark outside outer window FWD : BOOL:=0; // EPOS-Wort-2 Bit 04 --> 1 = Axis forwards BWD : BOOL:=0; // EPOS-Wort-2 Bit 05 --> 1 = Axis backwards SftSwMinAct : BOOL:=0; // EPOS-Wort-2 Bit 06 --> 1 = Software limit switch minus active SftSwPlsAct : BOOL:=0; // EPOS-Wort-2 Bit 07 --> 1 = Software limit switch plus active END_STRUCT;
         ZSW2 : Word := WORD#16#0000;   // ZSW2sxZSW2 : STRUCT Bit08 : BOOL:=0; // ZSW-Wort-2 Bit 08 --> Reserve GlbTrgReq : BOOL:=0; // ZSW-Wort-2 Bit 09 --> Global trigger request PulsEn : BOOL:=0; // ZSW-Wort-2 Bit 10 --> Pulses enabled MotSwOverAct : BOOL:=0; // ZSW-Wort-2 Bit 11 --> Motor switch over activ SlvZykBit0 : BOOL:=0; // ZSW-Wort-2 Bit 12 --> Slave - life bit 0 SlvZykBit1 : BOOL:=0; // ZSW-Wort-2 Bit 13 --> Slave - life bit 1 SlvZykBit2 : BOOL:=0; // ZSW-Wort-2 Bit 14 --> Slave - life bit 2 SlvZykBit3 : BOOL:=0; // ZSW-Wort-2 Bit 15 --> Slave - life bit 3 ActDDSBit0 : BOOL:=0; // ZSW-Wort-2 Bit 00 --> Active drive data set bit 0 ActDDSBit1 : BOOL:=0; // ZSW-Wort-2 Bit 01 --> Active drive data set bit 1 ActDDSBit2 : BOOL:=0; // ZSW-Wort-2 Bit 02 --> Active drive data set bit 2 ActDDSBit3 : BOOL:=0; // ZSW-Wort-2 Bit 03 --> Active drive data set bit 3 ActDDSBit4 : BOOL:=0; // ZSW-Wort-2 Bit 04 --> Active drive data set bit 4 CmdActRelBrk : BOOL:=0; // ZSW-Wort-2 Bit 05 --> Command "release holding break" active TrqContMode : BOOL:=0; // ZSW-Wort-2 Bit 06 --> Torque controlled mode ParkAxisAct : BOOL:=0; // ZSW-Wort-2 Bit 07 --> Parking axis activated END_STRUCT;
         NotUsed : Word := WORD#16#0000;   // Reserve
         Position : DWord := DWORD#16#0000_0000;   // Feedback of position
         Velocity : DWord := DWORD#16#0000_0000;   // Feedback of velocity
         ErrNr : Word := WORD#16#0000;   // Fault number
         WarnNr : Word := WORD#16#0000;   // Warning number
         Reserve : Word := WORD#16#0000;   // Reserve
      END_STRUCT;
   END_VAR
   VAR_TEMP
      piRetSFC : Int;   // Status for fault analysis
      piCount : Int;   // Freely available counter variable 3
      swSendBuf : Array[0..11] of Word;   // Send buffer
      swRecvBuf : Array[0..11] of Word;   // Receive buffer
   END_VAR
BEGIN

   //=============================================================================
   //SIEMENS AG
   //(c)Copyright 2019 All Rights Reserved
   //-----------------------------------------------------------------------------
   // Library: DriveLib
   // Tested with: -
   // Engineering: TIA Portal V15.1
   // Restrictions: -
   // Requirements: S7-1200 / S7-1500
   // Functionality: cyclic communication between a SINAMICS (Basic positioner)and a PLC
   //                If in HWConfig Std.TLG 111 is projected 12 PZD-words are exchanged
   //                in every bus cycle.
   //                The parametrisation of these words is described in the manual of the
   //                SINAMICS
   //=============================================================================

   // Betriebsart ermitteln
   IF #ModePos > #siModePosMax THEN

     #sbModePos := FALSE;
     #Error := True;
     #swStatus := 16#8202;
   ELSIF #ModePos < 1 THEN

     #sbModePos := FALSE;
     #Error := True;
     #swStatus := 16#8202;
   ELSE
     // Betriebsartenwechsel ist nur möglich, wenn die Achse nicht beschleunigt oder nicht verzögert 
     // und die Geschwindigkeit Null ist
     IF NOT #sbFWD AND NOT #sbBWD AND NOT #sbAccel AND NOT #sbDecel THEN

       #sbModePos := TRUE;
       #siModePos := #ModePos;

       // Fehler wieder zurücknehmen, wenn er mal ausgelöst wurde
       IF #swStatus = 16#8202 THEN
         #swStatus := 16#7002;
         #Error := False;
       END_IF;
     END_IF;
   END_IF;

   // Überprüfung der analogen Eingabewerte, ob sie innerhalb des möglichen Bereiches liegen
   // Geschwindigkeitsoverride (0% - 199%, 100% => W#16#4000)
   IF (#OverV < 0) OR (#OverV > 199) THEN
     #swStatus := 16#8203;
     #Error := True;
   ELSE
     // Geschwindigkeitsoverride in den Sendepuffer eintragen
     #sxSendBuf.OverrideV := INT_TO_WORD(REAL_TO_INT(16384.0 * (INT_TO_REAL(#OverV) / 100.0)));
   END_IF;

   // Beschleunigungsoverride (0% - 100%, 100% => W#16#4000)
   IF (#OverAcc < 0) OR (#OverAcc > 100) THEN
     #swStatus := 16#8203;
     #Error := True;
   ELSE
     // Beschleunigungsoverride in den Sendepuffer eintragen
     #sxSendBuf.OverrideA := INT_TO_WORD(REAL_TO_INT(16384.0 * (INT_TO_REAL(#OverAcc) / 100.0)));
   END_IF;

   // Verzögerungsoverride (0% - 100%, 100% => W#16#4000)
   IF (#OverDec < 0) OR (#OverDec > 100) THEN
     #swStatus := 16#8203;
     #Error := True;
   ELSE
     // Verzögerungsoverride in den Sendepuffer eintragen
     #sxSendBuf.OverrideD := INT_TO_WORD(REAL_TO_INT(16384.0 * (INT_TO_REAL(#OverDec) / 100.0)));
   END_IF;

   // Fehler wieder zurücknehmen, wenn er mal ausgelöst wurde
   IF NOT (#OverV < 0) AND NOT (#OverV > 199) AND NOT (#OverAcc < 0) AND NOT (#OverAcc > 100) AND
     NOT (#OverDec < 0) AND NOT (#OverDec > 100) THEN
     IF #swStatus = 16#8203 THEN
       #swStatus := 16#7002;
       #Error := False;
     END_IF;
   END_IF;

   // Positionssollwert
   // Positionssollwert in den Sendepuffer eintragen
   #sxSendBuf.Position := DINT_TO_DWORD(#Position);

   // Geschwindigkeitssollwert (Begrenzung / Überwachung
   // Geschwindigkeitssollwert in den Sendepuffer eintragen
   #sxSendBuf.Velocity := DINT_TO_DWORD(#Velocity);

   // Einschalten bzw. Ausschalten des Antriebes erkennen
   IF #EnableAxis AND NOT #sbOff1Edge AND NOT #sbBusy AND #sbModePos THEN
     #sbOff1 := True;
   END_IF;
   // Einschalten bzw. Ausschalten des Antriebes Flanke merken
   #sbOff1Edge := #EnableAxis AND NOT #sbBusy;

   // Einschaltflankenmerker wieder zurücksetzen
   IF NOT #EnableAxis THEN
     #sbOff1 := False;
   END_IF;

   // Fliegendes Referenzieren aktivieren erkennen
   IF #FlyRef AND NOT #sbRefTypEdge THEN
     #sbRefTyp := True;
   END_IF;
   // Fliegendes Referenzieren aktivieren Flanke merken
   #sbRefTypEdge := #FlyRef;

   // Fliegendes Referenzieren Flankenmerker wieder zurücksetzen
   IF NOT #FlyRef THEN
     #sbRefTyp := False;
     #siRefTypCyc := 0;
   END_IF;

   // Betriebsart aktivieren erkennen (RQ 3901129, RQ 4094299)
   IF #ExecuteMode AND NOT #sbExecuteEdge THEN
     #sbExecute := True;
     #siExecuteCyc := 0;
   ELSIF #ActMode <> #ModePos THEN
     #sbExecute := FALSE;
   ELSIF #siExecuteCyc > (2 * #siCycWait) THEN
     IF #ModePos <> 4 THEN
       #sbExecute := FALSE;
     ELSE
       IF #sxRecvBuf.ZSW1.%X11 OR NOT #ExecuteMode THEN
         #sbExecute := FALSE;
       END_IF;
     END_IF;
   ELSE
     ; // not used
   END_IF;

   IF #siExecuteCyc > 100 THEN
     #siExecuteCyc := 0;
   ELSE
     #siExecuteCyc := #siExecuteCyc + 1;
   END_IF;

   // Verfahrauftrag aktivieren Flanke merken
   #sbExecuteEdge := #ExecuteMode;

   // Betriebsart MDI / Sollwertdirektvorgabe Flanke merken
   (*IF #sxSendBuf.sxEPosSTW1.MdiStart AND NOT #sbMdiStartEdge THEN
             #sbMdiStart := True;
         END_IF;
         // Betriebsart MDI / Sollwertdirektvorgabe Flanke merken
         #sbMdiStartEdge := #sxSendBuf.sxEPosSTW1.MdiStart AND NOT #Busy;*)

   // Verfahrauftragflankenmerker wieder zurücksetzen
   (*IF NOT #sxSendBuf.sxEPosSTW1.MdiStart THEN
             #sbMdiStart := False;
             #siMdiStartCyc := 0;
         END_IF;*)

   IF #sxSendBuf.EPosSTW1.%X15 AND NOT #sbMdiStartEdge THEN
     #sbMdiStart := True;
   END_IF;
   // Betriebsart MDI / Sollwertdirektvorgabe Flanke merken
   #sbMdiStartEdge := #sxSendBuf.EPosSTW1.%X15 AND NOT #sbBusy;

   // Verfahrauftragflankenmerker wieder zurücksetzen
   IF NOT #sxSendBuf.EPosSTW1.%X15 THEN
     #sbMdiStart := False;
     #siMdiStartCyc := 0;
   END_IF;

   // Schreibdaten zusammenstellen
   // Steuerword STW1 für alle Betriebsart aufbereiten
   (*#sxSendBuf.sxSTW1.RejTrvTsk        := #RejTrvTsk;
         #sxSendBuf.sxSTW1.IntMStop         := #IntMStop;
         #sxSendBuf.sxSTW1.AckFault         := #AckFlt;*)

   #sxSendBuf.STW1.%X4 := #CancelTraversing;
   #sxSendBuf.STW1.%X5 := #IntermediateStop;
   #sxSendBuf.STW1.%X7 := #AckError;
   #sxSendBuf.STW1.%X1 := TRUE;
   #sxSendBuf.STW1.%X2 := TRUE;
   #sxSendBuf.STW1.%X3 := TRUE;
   #sxSendBuf.STW1.%X10 := TRUE;

   // Hauptbetriebsart "Positionieren / manueller Sollwertvorgabe (MDI)" 
   // Betriebsart "Positionieren Relativ positiv" oder "Positionieren Relativ negativ"
   IF (#siModePos = 1 AND #sbModePos) THEN

     // Antrieb einschalten
     //#sxSendBuf.sxSTW1.Off1 := #sbOff1;
     #sxSendBuf.STW1.%X0 := #sbOff1;

     // nicht verwendete Signale für den 1. Schritt und eventuell weitere Schritte
     (*#sxSendBuf.sxSTW1.Jog1          := False;
             #sxSendBuf.sxSTW1.Jog2          := False;
             #sxSendBuf.sxEPosSTW1.MdiTyp    := False;
             #sxSendBuf.sxEPosSTW1.MdiPos    := False;
             #sxSendBuf.sxEPosSTW1.MdiNeg    := False;
             #sxSendBuf.sxEPosSTW1.MdiSetup  := False;
             #sxSendBuf.sxEPosSTW2.SetRefPt  := False;
             #sxSendBuf.sxEPosSTW2.JogInc    := False;
             #sxSendBuf.sxEPosSTW2.RefStDi   := False;
             #sxSendBuf.sxSTW1.RefStart      := False;
             #sxSendBuf.sxEPosSTW2.RefTyp    := False;
             #sxSendBuf.sxEPosSTW1.MdiStart  := False;*)
     #sxSendBuf.STW1.%X8 := False;
     #sxSendBuf.STW1.%X9 := False;
     #sxSendBuf.EPosSTW1.%X8 := False;
     #sxSendBuf.EPosSTW1.%X9 := False;
     #sxSendBuf.EPosSTW1.%X10 := False;
     #sxSendBuf.EPosSTW1.%X14 := False;
     #sxSendBuf.EPosSTW2.%X1 := False;
     #sxSendBuf.EPosSTW2.%X5 := False;
     #sxSendBuf.EPosSTW2.%X9 := False;
     #sxSendBuf.STW1.%X11 := False;
     #sxSendBuf.EPosSTW2.%X8 := False;
     #sxSendBuf.EPosSTW1.%X15 := False;


     // Nach dem Einschalten des Antriebes, prüfen ob der Antrieb betriebsbereit, in Operation ohne Fehler und Warnung ist, 
     // dann die Betriebsart MDI / Sollwertvorgabe Start gesetzt werden
     IF #sbOff1 AND #sbReady AND #sbIOp AND NOT #sbFault THEN

       // Betriebsart MDI / Sollwertdirektvorgabe setzen
       //#sxSendBuf.sxEPosSTW1.MdiStart := True;
       #sxSendBuf.EPosSTW1.%X15 := True;

       // Positioniertyp auf relatives Positionieren stellen 
       //#sxSendBuf.sxEPosSTW1.MdiTyp := False;
       #sxSendBuf.EPosSTW1.%X8 := False;

       // die Richtungswahl für das Positionieren auf positive Richtung oder negative Richtung einstellen
       IF #Positive AND NOT #Negative THEN

         // positive Richtung
         //#sxSendBuf.sxEPosSTW1.MdiPos := True;
         #sxSendBuf.EPosSTW1.%X9 := True;

         // negative Richtung
         //#sxSendBuf.sxEPosSTW1.MdiNeg := False;
         #sxSendBuf.EPosSTW1.%X10 := False;

         // die Richtungswahl für das Positionieren auf negative Richtung einstellen                
       ELSIF NOT #Positive AND #Negative THEN

         // positive Richtung
         //#sxSendBuf.sxEPosSTW1.MdiPos := False;
         #sxSendBuf.EPosSTW1.%X9 := False;

         // negative Richtung
         //#sxSendBuf.sxEPosSTW1.MdiNeg := True;
         #sxSendBuf.EPosSTW1.%X10 := True;

         // die Richtungswahl für das Positionieren auf keine Richtung einstellen                
       ELSE

         // positive Richtung
         //#sxSendBuf.sxEPosSTW1.MdiPos := False;
         #sxSendBuf.EPosSTW1.%X9 := False;

         // negative Richtung
         //#sxSendBuf.sxEPosSTW1.MdiNeg := False;
         #sxSendBuf.EPosSTW1.%X10 := False;

       END_IF;

       // Nach dem Einschalten des Antriebes und dem Betriebsart MDI / Sollwertvorgabe starten, 
       // ein Paar Zyklen warten bevor die Flanke für die Sollwertübernahme MDI gesetzt werden kann
       IF #sbMdiStart AND (#siMdiStartCyc < #siCycWait) THEN
         #siMdiStartCyc := #siMdiStartCyc + 1;
       ELSE
         // Flanke Sollwertübernahme MDI
         //#sxSendBuf.sxSTW1.TrvStart := #Execute;
         #sxSendBuf.STW1.%X6 := #sbExecute;

       END_IF;

       // "Fliegendes Referentieren" aktivieren
       // "Fliegendes Referenzieren" erst nach Einschalten des Antriebes möglich
       IF #sbRefTyp THEN

         // Referenziertyp auf "Fliegendes Referenzieren" einstellen
         //#sxSendBuf.sxEPosSTW2.RefTyp := True;
         #sxSendBuf.EPosSTW2.%X8 := True;

         // Nach der Anwahl des Referenziertyps "Fliegendes Referenzieren", 
         // ein Zyklus später kann das Referenzieren gestartet
         IF (#siRefTypCyc = 0) THEN
           #siRefTypCyc := #siRefTypCyc + 1;
         ELSE
           // Referenzieren starten
           //#sxSendBuf.sxSTW1.RefStart := True;
           #sxSendBuf.STW1.%X11 := True;

         END_IF;
       END_IF;
     END_IF;

     // Betriebsart "Positionieren Absolut" oder "Positonieren Absolut positiv" oder "Positionieren Absolut negativ"
   ELSIF #siModePos = 2 AND #sbModePos THEN

     // Antrieb einschalten
     //#sxSendBuf.sxSTW1.Off1 := #sbOff1;
     #sxSendBuf.STW1.%X0 := #sbOff1;

     // nicht verwendete Signale für den 1. Schritt und eventuell weitere Schritte
     (*#sxSendBuf.sxSTW1.Jog1         := False;
             #sxSendBuf.sxSTW1.Jog2         := False;
             #sxSendBuf.sxEPosSTW1.MdiTyp   := False;
             #sxSendBuf.sxEPosSTW1.MdiPos   := False;
             #sxSendBuf.sxEPosSTW1.MdiNeg   := False;
             #sxSendBuf.sxEPosSTW1.MdiSetup := False;
             #sxSendBuf.sxEPosSTW2.SetRefPt := False;
             #sxSendBuf.sxEPosSTW2.JogInc   := False;
             #sxSendBuf.sxEPosSTW2.RefStDi  := False;
             #sxSendBuf.sxSTW1.RefStart     := False;
             #sxSendBuf.sxEPosSTW2.RefTyp   := False;
             #sxSendBuf.sxEPosSTW1.MdiStart := False;*)
     #sxSendBuf.STW1.%X8 := False;
     #sxSendBuf.STW1.%X9 := False;
     #sxSendBuf.EPosSTW1.%X8 := False;
     #sxSendBuf.EPosSTW1.%X9 := False;
     #sxSendBuf.EPosSTW1.%X10 := False;
     #sxSendBuf.EPosSTW1.%X14 := False;
     #sxSendBuf.EPosSTW2.%X1 := False;
     #sxSendBuf.EPosSTW2.%X5 := False;
     #sxSendBuf.EPosSTW2.%X9 := False;
     #sxSendBuf.STW1.%X11 := False;
     #sxSendBuf.EPosSTW2.%X8 := False;
     #sxSendBuf.EPosSTW1.%X15 := False;

     // Nach dem Einschalten des Antriebes, prüfen ob der Antrieb betriebsbereit, in Operation ohne Fehler und Warnung ist, 
     // dann die Betriebsart MDI / Sollwertvorgabe Start gesetzt werden
     IF #sbOff1 AND #sbReady AND #sbIOp AND NOT #sbFault THEN

       // Betriebsart MDI / Sollwertdirektvorgabe setzen
       //#sxSendBuf.sxEPosSTW1.MdiStart := True;
       #sxSendBuf.EPosSTW1.%X15 := True;

       // Positioniertyp auf absolutes Positionieren stellen 
       //#sxSendBuf.sxEPosSTW1.MdiTyp := True;
       #sxSendBuf.EPosSTW1.%X8 := True;

       // die Richtungswahl für das Positionieren auf positive Richtung oder negative Richtung einstellen
       IF #Positive AND NOT #Negative THEN

         // positive Richtung
         //#sxSendBuf.sxEPosSTW1.MdiPos := True;
         #sxSendBuf.EPosSTW1.%X9 := True;

         // negative Richtung
         //#sxSendBuf.sxEPosSTW1.MdiNeg := False;
         #sxSendBuf.EPosSTW1.%X10 := False;

         // die Richtungswahl für das Positionieren auf negative Richtung einstellen                
       ELSIF NOT #Positive AND #Negative THEN

         // positive Richtung
         //#sxSendBuf.sxEPosSTW1.MdiPos := False;
         #sxSendBuf.EPosSTW1.%X9 := False;

         // negative Richtung
         //#sxSendBuf.sxEPosSTW1.MdiNeg := True;
         #sxSendBuf.EPosSTW1.%X10 := True;

         // die Richtungswahl für das Positionieren auf keine Richtung einstellen                
       ELSE

         // positive Richtung
         //#sxSendBuf.sxEPosSTW1.MdiPos := False;
         #sxSendBuf.EPosSTW1.%X9 := False;

         // negative Richtung
         //#sxSendBuf.sxEPosSTW1.MdiNeg := False;
         #sxSendBuf.EPosSTW1.%X10 := False;

       END_IF;

       // Nach dem Einschalten des Antriebes und dem Betriebsart MDI / Sollwertvorgabe starten, 
       // ein Paar Zyklen warten bevor die Flanke für die Sollwertübernahme MDI gesetzt werden kann
       IF #sbMdiStart AND (#siMdiStartCyc < #siCycWait) THEN
         #siMdiStartCyc := #siMdiStartCyc + 1;
       ELSE
         // Flanke Sollwertübernahme MDI
         //#sxSendBuf.sxSTW1.TrvStart := #Execute;
         #sxSendBuf.STW1.%X6 := #sbExecute;

       END_IF;

       // "Fliegendes Referentieren" aktivieren
       // "Fliegendes Referenzieren" erst nach Einschalten des Antriebes möglich
       IF #sbRefTyp THEN

         // Referenziertyp auf "Fliegendes Referenzieren" einstellen
         //#sxSendBuf.sxEPosSTW2.RefTyp := True;
         #sxSendBuf.EPosSTW2.%X8 := True;

         // Nach der Anwahl des Referenziertyps "Fliegendes Referenzieren", 
         // ein Zyklus später kann das Referenzieren gestartet
         IF (#siRefTypCyc = 0) THEN
           #siRefTypCyc := #siRefTypCyc + 1;
         ELSE
           // Referenzieren starten
           //#sxSendBuf.sxSTW1.RefStart := True;
           #sxSendBuf.STW1.%X11 := True;

         END_IF;
       END_IF;
     END_IF;

     // Betriebsart "Positionieren als Einrichten positiv" oder "Positionieren als Einrichten negativ"
   ELSIF #siModePos = 3 AND #sbModePos THEN

     // Antrieb einschalten
     //#sxSendBuf.sxSTW1.Off1 := #sbOff1;
     #sxSendBuf.STW1.%X0 := #sbOff1;

     // nicht verwendete Signale für den 1. Schritt und eventuell weitere Schritte
     (*#sxSendBuf.sxSTW1.Jog1           := False;
             #sxSendBuf.sxSTW1.Jog2           := False;
             #sxSendBuf.sxEPosSTW1.MdiTyp     := False;
             #sxSendBuf.sxEPosSTW1.MdiPos     := False;
             #sxSendBuf.sxEPosSTW1.MdiNeg     := False;
             #sxSendBuf.sxEPosSTW1.MdiSetup   := False;
             #sxSendBuf.sxEPosSTW2.SetRefPt   := False;
             #sxSendBuf.sxEPosSTW2.JogInc     := False;
             #sxSendBuf.sxEPosSTW2.RefStDi    := False;
             #sxSendBuf.sxSTW1.RefStart       := False;
             #sxSendBuf.sxEPosSTW2.RefTyp     := False;
             #sxSendBuf.sxEPosSTW1.MdiStart   := False;*)
     #sxSendBuf.STW1.%X8 := False;
     #sxSendBuf.STW1.%X9 := False;
     #sxSendBuf.EPosSTW1.%X8 := False;
     #sxSendBuf.EPosSTW1.%X9 := False;
     #sxSendBuf.EPosSTW1.%X10 := False;
     #sxSendBuf.EPosSTW1.%X14 := False;
     #sxSendBuf.EPosSTW2.%X1 := False;
     #sxSendBuf.EPosSTW2.%X5 := False;
     #sxSendBuf.EPosSTW2.%X9 := False;
     #sxSendBuf.STW1.%X11 := False;
     #sxSendBuf.EPosSTW2.%X8 := False;
     #sxSendBuf.EPosSTW1.%X15 := False;

     // Nach dem Einschalten des Antriebes, prüfen ob der Antrieb betriebsbereit, in Operation ohne Fehler und Warnung ist, 
     // dann die Betriebsart MDI / Sollwertvorgabe Start gesetzt werden
     IF #sbOff1 AND #sbReady AND #sbIOp AND NOT #sbFault THEN

       // Betriebsart MDI / Sollwertdirektvorgabe setzen
       //#sxSendBuf.sxEPosSTW1.MdiStart := True;
       #sxSendBuf.EPosSTW1.%X15 := True;

       // Positioniertyp auf absolutes Positionieren stellen 
       //#sxSendBuf.sxEPosSTW1.MdiTyp := True;
       #sxSendBuf.EPosSTW1.%X8 := True;

       // die Anwahl für MDI Modus auf Einrichten einstellen
       //#sxSendBuf.sxEPosSTW1.MdiSetup := True;
       #sxSendBuf.EPosSTW1.%X14 := True;

       // die Richtungswahl für das Positionieren auf positive Richtung oder negative Richtung einstellen
       IF #Positive AND NOT #Negative THEN

         // positive Richtung
         //#sxSendBuf.sxEPosSTW1.MdiPos := True;
         #sxSendBuf.EPosSTW1.%X9 := True;

         // negative Richtung
         //#sxSendBuf.sxEPosSTW1.MdiNeg := False;
         #sxSendBuf.EPosSTW1.%X10 := False;

         // die Richtungswahl für das Positionieren auf negative Richtung einstellen                
       ELSIF NOT #Positive AND #Negative THEN

         // positive Richtung
         //#sxSendBuf.sxEPosSTW1.MdiPos := False;
         #sxSendBuf.EPosSTW1.%X9 := False;

         // negative Richtung
         //#sxSendBuf.sxEPosSTW1.MdiNeg := True;
         #sxSendBuf.EPosSTW1.%X10 := True;

         // die Richtungswahl für das Positionieren auf keine Richtung einstellen                
       ELSE

         // positive Richtung
         //#sxSendBuf.sxEPosSTW1.MdiPos := False;
         #sxSendBuf.EPosSTW1.%X9 := False;

         // negative Richtung
         //#sxSendBuf.sxEPosSTW1.MdiNeg := False;
         #sxSendBuf.EPosSTW1.%X10 := False;

       END_IF;

       // Nach dem Einschalten des Antriebes und dem Betriebsart MDI / Sollwertvorgabe starten, 
       // ein Paar Zyklen warten bevor die Flanke für die Sollwertübernahme MDI gesetzt werden kann
       IF #sbMdiStart AND (#siMdiStartCyc < #siCycWait) THEN
         #siMdiStartCyc := #siMdiStartCyc + 1;
       ELSE
         // Flanke Sollwertübernahme MDI
         //#sxSendBuf.sxSTW1.TrvStart := #Execute;
         #sxSendBuf.STW1.%X6 := #sbExecute;

       END_IF;

       // "Fliegendes Referentieren" aktivieren
       // "Fliegendes Referenzieren" erst nach Einschalten des Antriebes möglich
       IF #sbRefTyp THEN

         // Referenziertyp auf "Fliegendes Referenzieren" einstellen
         //#sxSendBuf.sxEPosSTW2.RefTyp := True;
         #sxSendBuf.EPosSTW2.%X8 := True;

         // Nach der Anwahl des Referenziertyps "Fliegendes Referenzieren", 
         // ein Zyklus später kann das Referenzieren gestartet
         IF (#siRefTypCyc = 0) THEN
           #siRefTypCyc := #siRefTypCyc + 1;
         ELSE
           // Referenzieren starten
           //#sxSendBuf.sxSTW1.RefStart := True;
           #sxSendBuf.STW1.%X11 := True;

         END_IF;
       END_IF;
     END_IF;

     // Hauptbetriebsart "Referenzieren" (Reference)
     // Betriebsart "Referenzieren - Referenzpunktfahrt positiv" oder "Referenzieren - Referenzpunktfahrt negativ"
   ELSIF #siModePos = 4 AND #sbModePos THEN

     // Antrieb einschalten
     //#sxSendBuf.sxSTW1.Off1 := #sbOff1;
     #sxSendBuf.STW1.%X0 := #sbOff1;

     // nicht verwendete Signale für den 1. Schritt und eventuell weitere Schritte
     (*#sxSendBuf.sxSTW1.Jog1         := False;
             #sxSendBuf.sxSTW1.Jog2         := False;
             #sxSendBuf.sxEPosSTW1.MdiStart := False;
             #sxSendBuf.sxEPosSTW2.SetRefPt := False;
             #sxSendBuf.sxEPosSTW2.JogInc   := False;
             #sxSendBuf.sxEPosSTW2.RefTyp   := False;
             #sxSendBuf.sxSTW1.RefStart     := False;
             #sxSendBuf.sxEPosSTW2.RefStDi  := False;*)
     #sxSendBuf.STW1.%X8 := False;
     #sxSendBuf.STW1.%X9 := False;
     #sxSendBuf.EPosSTW1.%X15 := False;
     #sxSendBuf.EPosSTW2.%X1 := False;
     #sxSendBuf.EPosSTW2.%X5 := False;
     #sxSendBuf.EPosSTW2.%X8 := False;
     #sxSendBuf.STW1.%X11 := False;
     #sxSendBuf.EPosSTW2.%X9 := False;

     // Nach dem Einschalten des Antriebes, prüfen ob der Antrieb betriebsbereit, in Operation ohne Fehler und Warnung ist, 
     // dann die Betriebsart MDI / Sollwertvorgabe Start gesetzt werden
     IF #sbOff1 AND #sbReady AND #sbIOp AND NOT #sbFault THEN

       // Referenzieren starten
       //#sxSendBuf.sxSTW1.RefStart := #Execute;
       #sxSendBuf.STW1.%X11 := #sbExecute;

       // die Richtungswahl für das Referenzpunktfahrt positiv einstellen
       IF #Positive AND NOT #Negative THEN

         // positive Referenzpunktfahrt
         //#sxSendBuf.sxEPosSTW2.RefStDi := False;
         #sxSendBuf.EPosSTW2.%X9 := False;

         // die Richtungswahl für das Referenzpunktfahrt negativ einstellen                
       ELSIF NOT #Positive AND #Negative THEN

         // negative Referenzpunktfahrt
         //#sxSendBuf.sxEPosSTW2.RefStDi := True;
         #sxSendBuf.EPosSTW2.%X9 := True;

       END_IF;
     END_IF;

     // Betriebsart "Referenzieren - Referenzpunkt setzen"
   ELSIF #siModePos = 5 AND #sbModePos THEN

     // Antrieb einschalten
     //#sxSendBuf.sxSTW1.Off1 := #sbOff1;
     #sxSendBuf.STW1.%X0 := #sbOff1;

     // nicht verwendete Signale für den 1. Schritt und eventuell weitere Schritte
     (*#sxSendBuf.sxSTW1.Jog1          := False;
             #sxSendBuf.sxSTW1.Jog2          := False;
             #sxSendBuf.sxSTW1.RefStart      := False;
             #sxSendBuf.sxEPosSTW1.MdiStart  := False;
             #sxSendBuf.sxEPosSTW2.JogInc    := False;
             #sxSendBuf.sxEPosSTW2.RefTyp    := False;
             #sxSendBuf.sxEPosSTW2.RefStDi   := False;
             #sxSendBuf.sxEPosSTW2.SetRefPt  := False;*)
     #sxSendBuf.STW1.%X8 := False;
     #sxSendBuf.STW1.%X9 := False;
     #sxSendBuf.STW1.%X11 := False;
     #sxSendBuf.EPosSTW1.%X15 := False;
     #sxSendBuf.EPosSTW2.%X5 := False;
     #sxSendBuf.EPosSTW2.%X8 := False;
     #sxSendBuf.EPosSTW2.%X9 := False;
     #sxSendBuf.EPosSTW2.%X1 := False;

     // Nach dem Einschalten des Antriebes, prüfen ob der Antrieb betriebsbereit, in Operation ohne Fehler und Warnung ist, 
     // dann die Betriebsart MDI / Sollwertvorgabe Start gesetzt werden
     IF NOT #sbFault THEN

       // Referenzpunktfahrt negativ
       //#sxSendBuf.sxEPosSTW2.SetRefPt := #Execute;
       #sxSendBuf.EPosSTW2.%X1 := #sbExecute;

     END_IF;

     // Hauptbetriebsart "Verfahrsätze" (Traversing Blocks)
   ELSIF #siModePos = 6 AND #sbModePos THEN

